   1:  PR[GP1:91,1] = PR[GP1:90,1] + -17.989;
   1:  PR[GP1:91,2] = PR[GP1:90,2] + 30.205;
   1:L PR[91] R[100]mm/sec CNT100;
   1:  PR[GP1:91,1] = PR[GP1:90,1] + -18.413;
   1:  PR[GP1:91,2] = PR[GP1:90,2] + 30.436;
   1:L PR[91] R[100]mm/sec CNT100;
   1:  PR[GP1:91,1] = PR[GP1:90,1] + -21.527;
   1:  PR[GP1:91,2] = PR[GP1:90,2] + 31.534;
   1:L PR[91] R[100]mm/sec CNT100;
   1:  PR[GP1:91,1] = PR[GP1:90,1] + -27.972;
   1:  PR[GP1:91,2] = PR[GP1:90,2] + 33.984;
   1:L PR[91] R[100]mm/sec CNT100;
   1:  PR[GP1:91,1] = PR[GP1:90,1] + -29.804;
   1:  PR[GP1:91,2] = PR[GP1:90,2] + 34.252;
   1:L PR[91] R[100]mm/sec CNT100;
   1:  PR[GP1:91,1] = PR[GP1:90,1] + -38.220;
   1:  PR[GP1:91,2] = PR[GP1:90,2] + 34.851;
   1:L PR[91] R[100]mm/sec CNT100;
   1:  PR[GP1:91,1] = PR[GP1:90,1] + -42.725;
   1:  PR[GP1:91,2] = PR[GP1:90,2] + 34.125;
   1:L PR[91] R[100]mm/sec CNT100;
   1:  PR[GP1:91,1] = PR[GP1:90,1] + -48.549;
   1:  PR[GP1:91,2] = PR[GP1:90,2] + 32.821;
   1:L PR[91] R[100]mm/sec CNT100;
   1:  PR[GP1:91,1] = PR[GP1:90,1] + -54.597;
   1:  PR[GP1:91,2] = PR[GP1:90,2] + 29.779;
   1:L PR[91] R[100]mm/sec CNT100;
   1:  PR[GP1:91,1] = PR[GP1:90,1] + -58.020;
   1:  PR[GP1:91,2] = PR[GP1:90,2] + 27.850;
   1:L PR[91] R[100]mm/sec CNT100;
   1:  PR[GP1:91,1] = PR[GP1:90,1] + -63.964;
   1:  PR[GP1:91,2] = PR[GP1:90,2] + 22.018;
   1:L PR[91] R[100]mm/sec CNT100;
   1:  PR[GP1:91,1] = PR[GP1:90,1] + -65.659;
   1:  PR[GP1:91,2] = PR[GP1:90,2] + 20.232;
   1:L PR[91] R[100]mm/sec CNT100;
   1:  PR[GP1:91,1] = PR[GP1:90,1] + -69.924;
   1:  PR[GP1:91,2] = PR[GP1:90,2] + 12.041;
   1:L PR[91] R[100]mm/sec CNT100;
   1:  PR[GP1:91,1] = PR[GP1:90,1] + -70.625;
   1:  PR[GP1:91,2] = PR[GP1:90,2] + 10.622;
   1:L PR[91] R[100]mm/sec CNT100;
   1:  PR[GP1:91,1] = PR[GP1:90,1] + -72.166;
   1:  PR[GP1:91,2] = PR[GP1:90,2] + 1.121;
   1:L PR[91] R[100]mm/sec CNT100;
   1:  PR[GP1:91,1] = PR[GP1:90,1] + -72.349;
   1:  PR[GP1:91,2] = PR[GP1:90,2] + 0.185;
   1:L PR[91] R[100]mm/sec CNT100;
   1:  PR[GP1:91,1] = PR[GP1:90,1] + -72.388;
   1:  PR[GP1:91,2] = PR[GP1:90,2] + -0.068;
   1:L PR[91] R[100]mm/sec CNT100;
   1:  PR[GP1:91,1] = PR[GP1:90,1] + -70.833;
   1:  PR[GP1:91,2] = PR[GP1:90,2] + -9.400;
   1:L PR[91] R[100]mm/sec CNT100;
   1:  PR[GP1:91,1] = PR[GP1:90,1] + -70.624;
   1:  PR[GP1:91,2] = PR[GP1:90,2] + -10.769;
   1:L PR[91] R[100]mm/sec CNT100;
   1:  PR[GP1:91,1] = PR[GP1:90,1] + -69.924;
   1:  PR[GP1:91,2] = PR[GP1:90,2] + -12.185;
   1:L PR[91] R[100]mm/sec CNT100;
   1:  PR[GP1:91,1] = PR[GP1:90,1] + -65.659;
   1:  PR[GP1:91,2] = PR[GP1:90,2] + -20.376;
   1:L PR[91] R[100]mm/sec CNT100;
   1:  PR[GP1:91,1] = PR[GP1:90,1] + -63.964;
   1:  PR[GP1:91,2] = PR[GP1:90,2] + -22.162;
   1:L PR[91] R[100]mm/sec CNT100;
   1:  PR[GP1:91,1] = PR[GP1:90,1] + -58.020;
   1:  PR[GP1:91,2] = PR[GP1:90,2] + -27.994;
   1:L PR[91] R[100]mm/sec CNT100;
   1:  PR[GP1:91,1] = PR[GP1:90,1] + -54.598;
   1:  PR[GP1:91,2] = PR[GP1:90,2] + -29.923;
   1:L PR[91] R[100]mm/sec CNT100;
   1:  PR[GP1:91,1] = PR[GP1:90,1] + -48.549;
   1:  PR[GP1:91,2] = PR[GP1:90,2] + -32.965;
   1:L PR[91] R[100]mm/sec CNT100;
   1:  PR[GP1:91,1] = PR[GP1:90,1] + -42.725;
   1:  PR[GP1:91,2] = PR[GP1:90,2] + -34.269;
   1:L PR[91] R[100]mm/sec CNT100;
   1:  PR[GP1:91,1] = PR[GP1:90,1] + -38.220;
   1:  PR[GP1:91,2] = PR[GP1:90,2] + -34.995;
   1:L PR[91] R[100]mm/sec CNT100;
   1:  PR[GP1:91,1] = PR[GP1:90,1] + -29.804;
   1:  PR[GP1:91,2] = PR[GP1:90,2] + -34.396;
   1:L PR[91] R[100]mm/sec CNT100;
   1:  PR[GP1:91,1] = PR[GP1:90,1] + -27.972;
   1:  PR[GP1:91,2] = PR[GP1:90,2] + -34.128;
   1:L PR[91] R[100]mm/sec CNT100;
   1:  PR[GP1:91,1] = PR[GP1:90,1] + -21.528;
   1:  PR[GP1:91,2] = PR[GP1:90,2] + -31.678;
   1:L PR[91] R[100]mm/sec CNT100;
   1:  PR[GP1:91,1] = PR[GP1:90,1] + -18.740;
   1:  PR[GP1:91,2] = PR[GP1:90,2] + -30.681;
   1:L PR[91] R[100]mm/sec CNT100;
   1:  PR[GP1:91,1] = PR[GP1:90,1] + -18.404;
   1:  PR[GP1:91,2] = PR[GP1:90,2] + -30.575;
   1:L PR[91] R[100]mm/sec CNT100;
   1:  PR[GP1:91,1] = PR[GP1:90,1] + -17.980;
   1:  PR[GP1:91,2] = PR[GP1:90,2] + -30.344;
   1:L PR[91] R[100]mm/sec CNT100;
   1:  PR[GP1:91,1] = PR[GP1:90,1] + -10.995;
   1:  PR[GP1:91,2] = PR[GP1:90,2] + -25.228;
   1:L PR[91] R[100]mm/sec CNT100;
   1:  PR[GP1:91,1] = PR[GP1:90,1] + -9.661;
   1:  PR[GP1:91,2] = PR[GP1:90,2] + -24.165;
   1:L PR[91] R[100]mm/sec CNT100;
   1:  PR[GP1:91,1] = PR[GP1:90,1] + -8.131;
   1:  PR[GP1:91,2] = PR[GP1:90,2] + -22.375;
   1:L PR[91] R[100]mm/sec CNT100;
   1:  PR[GP1:91,1] = PR[GP1:90,1] + -4.379;
   1:  PR[GP1:91,2] = PR[GP1:90,2] + -17.244;
   1:L PR[91] R[100]mm/sec CNT100;
   1:  PR[GP1:91,1] = PR[GP1:90,1] + -3.270;
   1:  PR[GP1:91,2] = PR[GP1:90,2] + -16.000;
   1:L PR[91] R[100]mm/sec CNT100;
   1:  PR[GP1:91,1] = PR[GP1:90,1] + -0.890;
   1:  PR[GP1:91,2] = PR[GP1:90,2] + -14.608;
   1:L PR[91] R[100]mm/sec CNT100;
   1:  PR[GP1:91,1] = PR[GP1:90,1] + 1.188;
   1:  PR[GP1:91,2] = PR[GP1:90,2] + -14.588;
   1:L PR[91] R[100]mm/sec CNT100;
   1:  PR[GP1:91,1] = PR[GP1:90,1] + 2.244;
   1:  PR[GP1:91,2] = PR[GP1:90,2] + -15.853;
   1:L PR[91] R[100]mm/sec CNT100;
   1:  PR[GP1:91,1] = PR[GP1:90,1] + 2.804;
   1:  PR[GP1:91,2] = PR[GP1:90,2] + -16.205;
   1:L PR[91] R[100]mm/sec CNT100;
   1:  PR[GP1:91,1] = PR[GP1:90,1] + 4.535;
   1:  PR[GP1:91,2] = PR[GP1:90,2] + -17.154;
   1:L PR[91] R[100]mm/sec CNT100;
   1:  PR[GP1:91,1] = PR[GP1:90,1] + 8.351;
   1:  PR[GP1:91,2] = PR[GP1:90,2] + -22.374;
   1:L PR[91] R[100]mm/sec CNT100;
   1:  PR[GP1:91,1] = PR[GP1:90,1] + 9.884;
   1:  PR[GP1:91,2] = PR[GP1:90,2] + -24.170;
   1:L PR[91] R[100]mm/sec CNT100;
   1:  PR[GP1:91,1] = PR[GP1:90,1] + 17.583;
   1:  PR[GP1:91,2] = PR[GP1:90,2] + -29.869;
   1:L PR[91] R[100]mm/sec CNT100;
   1:  PR[GP1:91,1] = PR[GP1:90,1] + 18.204;
   1:  PR[GP1:91,2] = PR[GP1:90,2] + -30.354;
   1:L PR[91] R[100]mm/sec CNT100;
   1:  PR[GP1:91,1] = PR[GP1:90,1] + 18.624;
   1:  PR[GP1:91,2] = PR[GP1:90,2] + -30.582;
   1:L PR[91] R[100]mm/sec CNT100;
   1:  PR[GP1:91,1] = PR[GP1:90,1] + 21.740;
   1:  PR[GP1:91,2] = PR[GP1:90,2] + -31.680;
   1:L PR[91] R[100]mm/sec CNT100;
   1:  PR[GP1:91,1] = PR[GP1:90,1] + 28.183;
   1:  PR[GP1:91,2] = PR[GP1:90,2] + -34.126;
   1:L PR[91] R[100]mm/sec CNT100;
   1:  PR[GP1:91,1] = PR[GP1:90,1] + 30.015;
   1:  PR[GP1:91,2] = PR[GP1:90,2] + -34.395;
   1:L PR[91] R[100]mm/sec CNT100;
   1:  PR[GP1:91,1] = PR[GP1:90,1] + 38.429;
   1:  PR[GP1:91,2] = PR[GP1:90,2] + -34.995;
   1:L PR[91] R[100]mm/sec CNT100;
   1:  PR[GP1:91,1] = PR[GP1:90,1] + 42.934;
   1:  PR[GP1:91,2] = PR[GP1:90,2] + -34.270;
   1:L PR[91] R[100]mm/sec CNT100;
   1:  PR[GP1:91,1] = PR[GP1:90,1] + 48.758;
   1:  PR[GP1:91,2] = PR[GP1:90,2] + -32.964;
   1:L PR[91] R[100]mm/sec CNT100;
   1:  PR[GP1:91,1] = PR[GP1:90,1] + 54.807;
   1:  PR[GP1:91,2] = PR[GP1:90,2] + -29.927;
   1:L PR[91] R[100]mm/sec CNT100;
   1:  PR[GP1:91,1] = PR[GP1:90,1] + 58.229;
   1:  PR[GP1:91,2] = PR[GP1:90,2] + -28.001;
   1:L PR[91] R[100]mm/sec CNT100;
   1:  PR[GP1:91,1] = PR[GP1:90,1] + 64.175;
   1:  PR[GP1:91,2] = PR[GP1:90,2] + -22.159;
   1:L PR[91] R[100]mm/sec CNT100;
   1:  PR[GP1:91,1] = PR[GP1:90,1] + 65.870;
   1:  PR[GP1:91,2] = PR[GP1:90,2] + -20.368;
   1:L PR[91] R[100]mm/sec CNT100;
   1:  PR[GP1:91,1] = PR[GP1:90,1] + 70.137;
   1:  PR[GP1:91,2] = PR[GP1:90,2] + -12.197;
   1:L PR[91] R[100]mm/sec CNT100;
   1:  PR[GP1:91,1] = PR[GP1:90,1] + 70.838;
   1:  PR[GP1:91,2] = PR[GP1:90,2] + -10.785;
   1:L PR[91] R[100]mm/sec CNT100;
   1:  PR[GP1:91,1] = PR[GP1:90,1] + 72.380;
   1:  PR[GP1:91,2] = PR[GP1:90,2] + -1.269;
   1:L PR[91] R[100]mm/sec CNT100;
   1:  PR[GP1:91,1] = PR[GP1:90,1] + 72.563;
   1:  PR[GP1:91,2] = PR[GP1:90,2] + -0.331;
   1:L PR[91] R[100]mm/sec CNT100;
   1:  PR[GP1:91,1] = PR[GP1:90,1] + 72.601;
   1:  PR[GP1:91,2] = PR[GP1:90,2] + -0.076;
   1:L PR[91] R[100]mm/sec CNT100;
   1:  PR[GP1:91,1] = PR[GP1:90,1] + 71.045;
   1:  PR[GP1:91,2] = PR[GP1:90,2] + 9.272;
   1:L PR[91] R[100]mm/sec CNT100;
   1:  PR[GP1:91,1] = PR[GP1:90,1] + 70.837;
   1:  PR[GP1:91,2] = PR[GP1:90,2] + 10.644;
   1:L PR[91] R[100]mm/sec CNT100;
   1:  PR[GP1:91,1] = PR[GP1:90,1] + 70.137;
   1:  PR[GP1:91,2] = PR[GP1:90,2] + 12.053;
   1:L PR[91] R[100]mm/sec CNT100;
   1:  PR[GP1:91,1] = PR[GP1:90,1] + 65.870;
   1:  PR[GP1:91,2] = PR[GP1:90,2] + 20.224;
   1:L PR[91] R[100]mm/sec CNT100;
   1:  PR[GP1:91,1] = PR[GP1:90,1] + 64.175;
   1:  PR[GP1:91,2] = PR[GP1:90,2] + 22.015;
   1:L PR[91] R[100]mm/sec CNT100;
   1:  PR[GP1:91,1] = PR[GP1:90,1] + 58.229;
   1:  PR[GP1:91,2] = PR[GP1:90,2] + 27.857;
   1:L PR[91] R[100]mm/sec CNT100;
   1:  PR[GP1:91,1] = PR[GP1:90,1] + 54.807;
   1:  PR[GP1:91,2] = PR[GP1:90,2] + 29.783;
   1:L PR[91] R[100]mm/sec CNT100;
   1:  PR[GP1:91,1] = PR[GP1:90,1] + 48.758;
   1:  PR[GP1:91,2] = PR[GP1:90,2] + 32.820;
   1:L PR[91] R[100]mm/sec CNT100;
   1:  PR[GP1:91,1] = PR[GP1:90,1] + 42.934;
   1:  PR[GP1:91,2] = PR[GP1:90,2] + 34.126;
   1:L PR[91] R[100]mm/sec CNT100;
   1:  PR[GP1:91,1] = PR[GP1:90,1] + 38.429;
   1:  PR[GP1:91,2] = PR[GP1:90,2] + 34.851;
   1:L PR[91] R[100]mm/sec CNT100;
   1:  PR[GP1:91,1] = PR[GP1:90,1] + 30.015;
   1:  PR[GP1:91,2] = PR[GP1:90,2] + 34.251;
   1:L PR[91] R[100]mm/sec CNT100;
   1:  PR[GP1:91,1] = PR[GP1:90,1] + 28.183;
   1:  PR[GP1:91,2] = PR[GP1:90,2] + 33.982;
   1:L PR[91] R[100]mm/sec CNT100;
   1:  PR[GP1:91,1] = PR[GP1:90,1] + 21.741;
   1:  PR[GP1:91,2] = PR[GP1:90,2] + 31.536;
   1:L PR[91] R[100]mm/sec CNT100;
   1:  PR[GP1:91,1] = PR[GP1:90,1] + 18.953;
   1:  PR[GP1:91,2] = PR[GP1:90,2] + 30.540;
   1:L PR[91] R[100]mm/sec CNT100;
   1:  PR[GP1:91,1] = PR[GP1:90,1] + 18.616;
   1:  PR[GP1:91,2] = PR[GP1:90,2] + 30.434;
   1:L PR[91] R[100]mm/sec CNT100;
   1:  PR[GP1:91,1] = PR[GP1:90,1] + 18.196;
   1:  PR[GP1:91,2] = PR[GP1:90,2] + 30.205;
   1:L PR[91] R[100]mm/sec CNT100;
   1:  PR[GP1:91,1] = PR[GP1:90,1] + 11.213;
   1:  PR[GP1:91,2] = PR[GP1:90,2] + 25.087;
   1:L PR[91] R[100]mm/sec CNT100;
   1:  PR[GP1:91,1] = PR[GP1:90,1] + 9.890;
   1:  PR[GP1:91,2] = PR[GP1:90,2] + 24.034;
   1:L PR[91] R[100]mm/sec CNT100;
   1:  PR[GP1:91,1] = PR[GP1:90,1] + 8.351;
   1:  PR[GP1:91,2] = PR[GP1:90,2] + 22.230;
   1:L PR[91] R[100]mm/sec CNT100;
   1:  PR[GP1:91,1] = PR[GP1:90,1] + 4.595;
   1:  PR[GP1:91,2] = PR[GP1:90,2] + 17.092;
   1:L PR[91] R[100]mm/sec CNT100;
   1:  PR[GP1:91,1] = PR[GP1:90,1] + 3.455;
   1:  PR[GP1:91,2] = PR[GP1:90,2] + 15.837;
   1:L PR[91] R[100]mm/sec CNT100;
   1:  PR[GP1:91,1] = PR[GP1:90,1] + 1.069;
   1:  PR[GP1:91,2] = PR[GP1:90,2] + 14.445;
   1:L PR[91] R[100]mm/sec CNT100;
   1:  PR[GP1:91,1] = PR[GP1:90,1] + -0.890;
   1:  PR[GP1:91,2] = PR[GP1:90,2] + 14.464;
   1:L PR[91] R[100]mm/sec CNT100;
   1:  ! -- Layer/Ebene 55 -- !;
   1:  PR[91] = PR[90];
   1:  PR[GP1:91,1] = PR[GP1:90,1] + -3.388;
   1:  PR[GP1:91,2] = PR[GP1:90,2] + 16.407;
   1:  PR[GP1:91,3] = PR[GP1:90,3] + 33.855;
   1:L PR[91] R[100]mm/sec CNT100;
   1:  PR[GP1:91,1] = PR[GP1:90,1] + -4.446;
   1:  PR[GP1:91,2] = PR[GP1:90,2] + 17.549;
   1:L PR[91] R[100]mm/sec CNT100;
   1:  PR[GP1:91,1] = PR[GP1:90,1] + -4.455;
   1:  PR[GP1:91,2] = PR[GP1:90,2] + 17.629;
   1:L PR[91] R[100]mm/sec CNT100;
   1:  PR[GP1:91,1] = PR[GP1:90,1] + -7.518;
   1:  PR[GP1:91,2] = PR[GP1:90,2] + 21.818;
   1:L PR[91] R[100]mm/sec CNT100;
   1:  PR[GP1:91,1] = PR[GP1:90,1] + -9.459;
   1:  PR[GP1:91,2] = PR[GP1:90,2] + 24.089;
   1:L PR[91] R[100]mm/sec CNT100;
   1:  PR[GP1:91,1] = PR[GP1:90,1] + -16.227;
   1:  PR[GP1:91,2] = PR[GP1:90,2] + 29.096;
   1:L PR[91] R[100]mm/sec CNT100;
   1:  PR[GP1:91,1] = PR[GP1:90,1] + -17.485;
   1:  PR[GP1:91,2] = PR[GP1:90,2] + 30.078;
   1:L PR[91] R[100]mm/sec CNT100;
   1:  PR[GP1:91,1] = PR[GP1:90,1] + -18.396;
   1:  PR[GP1:91,2] = PR[GP1:90,2] + 30.575;
   1:L PR[91] R[100]mm/sec CNT100;
   1:  PR[GP1:91,1] = PR[GP1:90,1] + -24.522;
   1:  PR[GP1:91,2] = PR[GP1:90,2] + 32.735;
   1:L PR[91] R[100]mm/sec CNT100;
   1:  PR[GP1:91,1] = PR[GP1:90,1] + -28.037;
   1:  PR[GP1:91,2] = PR[GP1:90,2] + 34.071;
   1:L PR[91] R[100]mm/sec CNT100;
   1:  PR[GP1:91,1] = PR[GP1:90,1] + -29.004;
   1:  PR[GP1:91,2] = PR[GP1:90,2] + 34.213;
   1:L PR[91] R[100]mm/sec CNT100;
   1:  PR[GP1:91,1] = PR[GP1:90,1] + -38.254;
   1:  PR[GP1:91,2] = PR[GP1:90,2] + 34.871;
   1:L PR[91] R[100]mm/sec CNT100;
   1:  PR[GP1:91,1] = PR[GP1:90,1] + -41.956;
   1:  PR[GP1:91,2] = PR[GP1:90,2] + 34.274;
   1:L PR[91] R[100]mm/sec CNT100;
   1:  PR[GP1:91,1] = PR[GP1:90,1] + -48.542;
   1:  PR[GP1:91,2] = PR[GP1:90,2] + 32.799;
   1:L PR[91] R[100]mm/sec CNT100;
   1:  PR[GP1:91,1] = PR[GP1:90,1] + -53.920;
   1:  PR[GP1:91,2] = PR[GP1:90,2] + 30.095;
   1:L PR[91] R[100]mm/sec CNT100;
   1:  PR[GP1:91,1] = PR[GP1:90,1] + -57.970;
   1:  PR[GP1:91,2] = PR[GP1:90,2] + 27.812;
   1:L PR[91] R[100]mm/sec CNT100;
   1:  PR[GP1:91,1] = PR[GP1:90,1] + -63.421;
   1:  PR[GP1:91,2] = PR[GP1:90,2] + 22.463;
   1:L PR[91] R[100]mm/sec CNT100;
   1:  PR[GP1:91,1] = PR[GP1:90,1] + -65.574;
   1:  PR[GP1:91,2] = PR[GP1:90,2] + 20.196;
   1:L PR[91] R[100]mm/sec CNT100;
   1:  PR[GP1:91,1] = PR[GP1:90,1] + -69.543;
   1:  PR[GP1:91,2] = PR[GP1:90,2] + 12.572;
   1:L PR[91] R[100]mm/sec CNT100;
   1:  PR[GP1:91,1] = PR[GP1:90,1] + -70.517;
   1:  PR[GP1:91,2] = PR[GP1:90,2] + 10.601;
   1:L PR[91] R[100]mm/sec CNT100;
   1:  PR[GP1:91,1] = PR[GP1:90,1] + -71.962;
   1:  PR[GP1:91,2] = PR[GP1:90,2] + 1.695;
   1:L PR[91] R[100]mm/sec CNT100;
   1:  PR[GP1:91,1] = PR[GP1:90,1] + -72.133;
   1:  PR[GP1:91,2] = PR[GP1:90,2] + 0.818;
   1:L PR[91] R[100]mm/sec CNT100;
   1:  PR[GP1:91,1] = PR[GP1:90,1] + -72.269;
   1:  PR[GP1:91,2] = PR[GP1:90,2] + -0.068;
   1:L PR[91] R[100]mm/sec CNT100;
   1:  PR[GP1:91,1] = PR[GP1:90,1] + -70.806;
   1:  PR[GP1:91,2] = PR[GP1:90,2] + -8.846;
   1:L PR[91] R[100]mm/sec CNT100;
   1:  PR[GP1:91,1] = PR[GP1:90,1] + -70.516;
   1:  PR[GP1:91,2] = PR[GP1:90,2] + -10.748;
   1:L PR[91] R[100]mm/sec CNT100;
   1:  PR[GP1:91,1] = PR[GP1:90,1] + -69.543;
   1:  PR[GP1:91,2] = PR[GP1:90,2] + -12.716;
   1:L PR[91] R[100]mm/sec CNT100;
   1:  PR[GP1:91,1] = PR[GP1:90,1] + -65.574;
   1:  PR[GP1:91,2] = PR[GP1:90,2] + -20.340;
   1:L PR[91] R[100]mm/sec CNT100;
   1:  PR[GP1:91,1] = PR[GP1:90,1] + -63.421;
   1:  PR[GP1:91,2] = PR[GP1:90,2] + -22.607;
   1:L PR[91] R[100]mm/sec CNT100;
   1:  PR[GP1:91,1] = PR[GP1:90,1] + -57.970;
   1:  PR[GP1:91,2] = PR[GP1:90,2] + -27.956;
   1:L PR[91] R[100]mm/sec CNT100;
   1:  PR[GP1:91,1] = PR[GP1:90,1] + -53.920;
   1:  PR[GP1:91,2] = PR[GP1:90,2] + -30.239;
   1:L PR[91] R[100]mm/sec CNT100;
   1:  PR[GP1:91,1] = PR[GP1:90,1] + -48.542;
   1:  PR[GP1:91,2] = PR[GP1:90,2] + -32.943;
   1:L PR[91] R[100]mm/sec CNT100;
   1:  PR[GP1:91,1] = PR[GP1:90,1] + -41.956;
   1:  PR[GP1:91,2] = PR[GP1:90,2] + -34.418;
   1:L PR[91] R[100]mm/sec CNT100;
   1:  PR[GP1:91,1] = PR[GP1:90,1] + -38.254;
   1:  PR[GP1:91,2] = PR[GP1:90,2] + -35.015;
   1:L PR[91] R[100]mm/sec CNT100;
   1:  PR[GP1:91,1] = PR[GP1:90,1] + -29.004;
   1:  PR[GP1:91,2] = PR[GP1:90,2] + -34.357;
   1:L PR[91] R[100]mm/sec CNT100;
   1:  PR[GP1:91,1] = PR[GP1:90,1] + -28.037;
   1:  PR[GP1:91,2] = PR[GP1:90,2] + -34.215;
   1:L PR[91] R[100]mm/sec CNT100;
   1:  PR[GP1:91,1] = PR[GP1:90,1] + -24.523;
   1:  PR[GP1:91,2] = PR[GP1:90,2] + -32.879;
   1:L PR[91] R[100]mm/sec CNT100;
   1:  PR[GP1:91,1] = PR[GP1:90,1] + -19.087;
   1:  PR[GP1:91,2] = PR[GP1:90,2] + -30.934;
   1:L PR[91] R[100]mm/sec CNT100;
   1:  PR[GP1:91,1] = PR[GP1:90,1] + -18.387;
   1:  PR[GP1:91,2] = PR[GP1:90,2] + -30.714;
   1:L PR[91] R[100]mm/sec CNT100;
   1:  PR[GP1:91,1] = PR[GP1:90,1] + -17.476;
   1:  PR[GP1:91,2] = PR[GP1:90,2] + -30.217;
   1:L PR[91] R[100]mm/sec CNT100;
   1:  PR[GP1:91,1] = PR[GP1:90,1] + -11.167;
   1:  PR[GP1:91,2] = PR[GP1:90,2] + -25.597;
   1:L PR[91] R[100]mm/sec CNT100;
   1:  PR[GP1:91,1] = PR[GP1:90,1] + -9.466;
   1:  PR[GP1:91,2] = PR[GP1:90,2] + -24.241;
   1:L PR[91] R[100]mm/sec CNT100;
   1:  PR[GP1:91,1] = PR[GP1:90,1] + -7.518;
   1:  PR[GP1:91,2] = PR[GP1:90,2] + -21.962;
   1:L PR[91] R[100]mm/sec CNT100;
   1:  PR[GP1:91,1] = PR[GP1:90,1] + -4.344;
   1:  PR[GP1:91,2] = PR[GP1:90,2] + -17.621;
   1:L PR[91] R[100]mm/sec CNT100;
   1:  PR[GP1:91,1] = PR[GP1:90,1] + -3.393;
   1:  PR[GP1:91,2] = PR[GP1:90,2] + -16.554;
   1:L PR[91] R[100]mm/sec CNT100;
   1:  PR[GP1:91,1] = PR[GP1:90,1] + -0.787;
   1:  PR[GP1:91,2] = PR[GP1:90,2] + -15.030;
   1:L PR[91] R[100]mm/sec CNT100;
   1:  PR[GP1:91,1] = PR[GP1:90,1] + 1.090;
   1:  PR[GP1:91,2] = PR[GP1:90,2] + -15.011;
   1:L PR[91] R[100]mm/sec CNT100;
   1:  PR[GP1:91,1] = PR[GP1:90,1] + 2.030;
   1:  PR[GP1:91,2] = PR[GP1:90,2] + -16.138;
   1:L PR[91] R[100]mm/sec CNT100;
   1:  PR[GP1:91,1] = PR[GP1:90,1] + 2.509;
   1:  PR[GP1:91,2] = PR[GP1:90,2] + -16.440;
   1:L PR[91] R[100]mm/sec CNT100;
   1:  PR[GP1:91,1] = PR[GP1:90,1] + 4.501;
   1:  PR[GP1:91,2] = PR[GP1:90,2] + -17.531;
   1:L PR[91] R[100]mm/sec CNT100;
   1:  PR[GP1:91,1] = PR[GP1:90,1] + 7.740;
   1:  PR[GP1:91,2] = PR[GP1:90,2] + -21.961;
   1:L PR[91] R[100]mm/sec CNT100;
   1:  PR[GP1:91,1] = PR[GP1:90,1] + 9.693;
   1:  PR[GP1:91,2] = PR[GP1:90,2] + -24.250;
   1:L PR[91] R[100]mm/sec CNT100;
   1:  PR[GP1:91,1] = PR[GP1:90,1] + 16.456;
   1:  PR[GP1:91,2] = PR[GP1:90,2] + -29.256;
   1:L PR[91] R[100]mm/sec CNT100;
   1:  PR[GP1:91,1] = PR[GP1:90,1] + 17.702;
   1:  PR[GP1:91,2] = PR[GP1:90,2] + -30.229;
   1:L PR[91] R[100]mm/sec CNT100;
   1:  PR[GP1:91,1] = PR[GP1:90,1] + 18.606;
   1:  PR[GP1:91,2] = PR[GP1:90,2] + -30.721;
   1:L PR[91] R[100]mm/sec CNT100;
   1:  PR[GP1:91,1] = PR[GP1:90,1] + 24.735;
   1:  PR[GP1:91,2] = PR[GP1:90,2] + -32.879;
   1:L PR[91] R[100]mm/sec CNT100;
   1:  PR[GP1:91,1] = PR[GP1:90,1] + 28.250;
   1:  PR[GP1:91,2] = PR[GP1:90,2] + -34.213;
   1:L PR[91] R[100]mm/sec CNT100;
   1:  PR[GP1:91,1] = PR[GP1:90,1] + 29.217;
   1:  PR[GP1:91,2] = PR[GP1:90,2] + -34.355;
   1:L PR[91] R[100]mm/sec CNT100;
   1:  PR[GP1:91,1] = PR[GP1:90,1] + 38.464;
   1:  PR[GP1:91,2] = PR[GP1:90,2] + -35.015;
   1:L PR[91] R[100]mm/sec CNT100;
   1:  PR[GP1:91,1] = PR[GP1:90,1] + 42.166;
   1:  PR[GP1:91,2] = PR[GP1:90,2] + -34.419;
   1:L PR[91] R[100]mm/sec CNT100;
   1:  PR[GP1:91,1] = PR[GP1:90,1] + 48.751;
   1:  PR[GP1:91,2] = PR[GP1:90,2] + -32.942;
   1:L PR[91] R[100]mm/sec CNT100;
   1:  PR[GP1:91,1] = PR[GP1:90,1] + 54.129;
   1:  PR[GP1:91,2] = PR[GP1:90,2] + -30.242;
   1:L PR[91] R[100]mm/sec CNT100;
   1:  PR[GP1:91,1] = PR[GP1:90,1] + 58.179;
   1:  PR[GP1:91,2] = PR[GP1:90,2] + -27.963;
   1:L PR[91] R[100]mm/sec CNT100;
   1:  PR[GP1:91,1] = PR[GP1:90,1] + 63.632;
   1:  PR[GP1:91,2] = PR[GP1:90,2] + -22.606;
   1:L PR[91] R[100]mm/sec CNT100;
   1:  PR[GP1:91,1] = PR[GP1:90,1] + 65.785;
   1:  PR[GP1:91,2] = PR[GP1:90,2] + -20.331;
   1:L PR[91] R[100]mm/sec CNT100;
   1:  PR[GP1:91,1] = PR[GP1:90,1] + 69.756;
   1:  PR[GP1:91,2] = PR[GP1:90,2] + -12.726;
   1:L PR[91] R[100]mm/sec CNT100;
   1:  PR[GP1:91,1] = PR[GP1:90,1] + 70.730;
   1:  PR[GP1:91,2] = PR[GP1:90,2] + -10.765;
   1:L PR[91] R[100]mm/sec CNT100;
   1:  PR[GP1:91,1] = PR[GP1:90,1] + 72.175;
   1:  PR[GP1:91,2] = PR[GP1:90,2] + -1.845;
   1:L PR[91] R[100]mm/sec CNT100;
   1:  PR[GP1:91,1] = PR[GP1:90,1] + 72.346;
   1:  PR[GP1:91,2] = PR[GP1:90,2] + -0.965;
   1:L PR[91] R[100]mm/sec CNT100;
   1:  PR[GP1:91,1] = PR[GP1:90,1] + 72.482;
   1:  PR[GP1:91,2] = PR[GP1:90,2] + -0.076;
   1:L PR[91] R[100]mm/sec CNT100;
   1:  PR[GP1:91,1] = PR[GP1:90,1] + 71.019;
   1:  PR[GP1:91,2] = PR[GP1:90,2] + 8.717;
   1:L PR[91] R[100]mm/sec CNT100;
   1:  PR[GP1:91,1] = PR[GP1:90,1] + 70.728;
   1:  PR[GP1:91,2] = PR[GP1:90,2] + 10.624;
   1:L PR[91] R[100]mm/sec CNT100;
   1:  PR[GP1:91,1] = PR[GP1:90,1] + 69.756;
   1:  PR[GP1:91,2] = PR[GP1:90,2] + 12.582;
   1:L PR[91] R[100]mm/sec CNT100;
   1:  PR[GP1:91,1] = PR[GP1:90,1] + 65.785;
   1:  PR[GP1:91,2] = PR[GP1:90,2] + 20.187;
   1:L PR[91] R[100]mm/sec CNT100;
   1:  PR[GP1:91,1] = PR[GP1:90,1] + 63.632;
   1:  PR[GP1:91,2] = PR[GP1:90,2] + 22.462;
   1:L PR[91] R[100]mm/sec CNT100;
   1:  PR[GP1:91,1] = PR[GP1:90,1] + 58.179;
   1:  PR[GP1:91,2] = PR[GP1:90,2] + 27.819;
   1:L PR[91] R[100]mm/sec CNT100;
   1:  PR[GP1:91,1] = PR[GP1:90,1] + 54.129;
   1:  PR[GP1:91,2] = PR[GP1:90,2] + 30.098;
   1:L PR[91] R[100]mm/sec CNT100;
   1:  PR[GP1:91,1] = PR[GP1:90,1] + 48.751;
   1:  PR[GP1:91,2] = PR[GP1:90,2] + 32.798;
   1:L PR[91] R[100]mm/sec CNT100;
   1:  PR[GP1:91,1] = PR[GP1:90,1] + 42.166;
   1:  PR[GP1:91,2] = PR[GP1:90,2] + 34.275;
   1:L PR[91] R[100]mm/sec CNT100;
   1:  PR[GP1:91,1] = PR[GP1:90,1] + 38.464;
   1:  PR[GP1:91,2] = PR[GP1:90,2] + 34.871;
   1:L PR[91] R[100]mm/sec CNT100;
   1:  PR[GP1:91,1] = PR[GP1:90,1] + 29.217;
   1:  PR[GP1:91,2] = PR[GP1:90,2] + 34.211;
   1:L PR[91] R[100]mm/sec CNT100;
   1:  PR[GP1:91,1] = PR[GP1:90,1] + 28.250;
   1:  PR[GP1:91,2] = PR[GP1:90,2] + 34.069;
   1:L PR[91] R[100]mm/sec CNT100;
   1:  PR[GP1:91,1] = PR[GP1:90,1] + 24.736;
   1:  PR[GP1:91,2] = PR[GP1:90,2] + 32.735;
   1:L PR[91] R[100]mm/sec CNT100;
   1:  PR[GP1:91,1] = PR[GP1:90,1] + 19.300;
   1:  PR[GP1:91,2] = PR[GP1:90,2] + 30.793;
   1:L PR[91] R[100]mm/sec CNT100;
   1:  PR[GP1:91,1] = PR[GP1:90,1] + 18.598;
   1:  PR[GP1:91,2] = PR[GP1:90,2] + 30.572;
   1:L PR[91] R[100]mm/sec CNT100;
   1:  PR[GP1:91,1] = PR[GP1:90,1] + 17.694;
   1:  PR[GP1:91,2] = PR[GP1:90,2] + 30.080;
   1:L PR[91] R[100]mm/sec CNT100;
   1:  PR[GP1:91,1] = PR[GP1:90,1] + 11.387;
   1:  PR[GP1:91,2] = PR[GP1:90,2] + 25.457;
   1:L PR[91] R[100]mm/sec CNT100;
   1:  PR[GP1:91,1] = PR[GP1:90,1] + 9.700;
   1:  PR[GP1:91,2] = PR[GP1:90,2] + 24.114;
   1:L PR[91] R[100]mm/sec CNT100;
   1:  PR[GP1:91,1] = PR[GP1:90,1] + 7.740;
   1:  PR[GP1:91,2] = PR[GP1:90,2] + 21.817;
   1:L PR[91] R[100]mm/sec CNT100;
   1:  PR[GP1:91,1] = PR[GP1:90,1] + 4.561;
   1:  PR[GP1:91,2] = PR[GP1:90,2] + 17.469;
   1:L PR[91] R[100]mm/sec CNT100;
   1:  PR[GP1:91,1] = PR[GP1:90,1] + 3.583;
   1:  PR[GP1:91,2] = PR[GP1:90,2] + 16.393;
   1:L PR[91] R[100]mm/sec CNT100;
   1:  PR[GP1:91,1] = PR[GP1:90,1] + 0.971;
   1:  PR[GP1:91,2] = PR[GP1:90,2] + 14.869;
   1:L PR[91] R[100]mm/sec CNT100;
   1:  PR[GP1:91,1] = PR[GP1:90,1] + -0.787;
   1:  PR[GP1:91,2] = PR[GP1:90,2] + 14.886;
   1:L PR[91] R[100]mm/sec CNT100;
   1:  ! -- Layer/Ebene 56 -- !;
   1:  PR[91] = PR[90];
   1:  PR[GP1:91,1] = PR[GP1:90,1] + -3.510;
   1:  PR[GP1:91,2] = PR[GP1:90,2] + 16.961;
   1:  PR[GP1:91,3] = PR[GP1:90,3] + 34.465;
   1:L PR[91] R[100]mm/sec CNT100;
   1:  PR[GP1:91,1] = PR[GP1:90,1] + -4.411;
   1:  PR[GP1:91,2] = PR[GP1:90,2] + 17.933;
   1:L PR[91] R[100]mm/sec CNT100;
   1:  PR[GP1:91,1] = PR[GP1:90,1] + -4.420;
   1:  PR[GP1:91,2] = PR[GP1:90,2] + 18.006;
   1:L PR[91] R[100]mm/sec CNT100;
   1:  PR[GP1:91,1] = PR[GP1:90,1] + -6.905;
   1:  PR[GP1:91,2] = PR[GP1:90,2] + 21.405;
   1:L PR[91] R[100]mm/sec CNT100;
   1:  PR[GP1:91,1] = PR[GP1:90,1] + -9.264;
   1:  PR[GP1:91,2] = PR[GP1:90,2] + 24.165;
   1:L PR[91] R[100]mm/sec CNT100;
   1:  PR[GP1:91,1] = PR[GP1:90,1] + -15.093;
   1:  PR[GP1:91,2] = PR[GP1:90,2] + 28.477;
   1:L PR[91] R[100]mm/sec CNT100;
   1:  PR[GP1:91,1] = PR[GP1:90,1] + -16.981;
   1:  PR[GP1:91,2] = PR[GP1:90,2] + 29.951;
   1:L PR[91] R[100]mm/sec CNT100;
   1:  PR[GP1:91,1] = PR[GP1:90,1] + -18.379;
   1:  PR[GP1:91,2] = PR[GP1:90,2] + 30.714;
   1:L PR[91] R[100]mm/sec CNT100;
   1:  PR[GP1:91,1] = PR[GP1:90,1] + -27.518;
   1:  PR[GP1:91,2] = PR[GP1:90,2] + 33.936;
   1:L PR[91] R[100]mm/sec CNT100;
   1:  PR[GP1:91,1] = PR[GP1:90,1] + -28.103;
   1:  PR[GP1:91,2] = PR[GP1:90,2] + 34.158;
   1:L PR[91] R[100]mm/sec CNT100;
   1:  PR[GP1:91,1] = PR[GP1:90,1] + -28.204;
   1:  PR[GP1:91,2] = PR[GP1:90,2] + 34.173;
   1:L PR[91] R[100]mm/sec CNT100;
   1:  PR[GP1:91,1] = PR[GP1:90,1] + -38.288;
   1:  PR[GP1:91,2] = PR[GP1:90,2] + 34.890;
   1:L PR[91] R[100]mm/sec CNT100;
   1:  PR[GP1:91,1] = PR[GP1:90,1] + -41.188;
   1:  PR[GP1:91,2] = PR[GP1:90,2] + 34.423;
   1:L PR[91] R[100]mm/sec CNT100;
   1:  PR[GP1:91,1] = PR[GP1:90,1] + -48.534;
   1:  PR[GP1:91,2] = PR[GP1:90,2] + 32.778;
   1:L PR[91] R[100]mm/sec CNT100;
   1:  PR[GP1:91,1] = PR[GP1:90,1] + -53.242;
   1:  PR[GP1:91,2] = PR[GP1:90,2] + 30.410;
   1:L PR[91] R[100]mm/sec CNT100;
   1:  PR[GP1:91,1] = PR[GP1:90,1] + -57.919;
   1:  PR[GP1:91,2] = PR[GP1:90,2] + 27.773;
   1:L PR[91] R[100]mm/sec CNT100;
   1:  PR[GP1:91,1] = PR[GP1:90,1] + -62.878;
   1:  PR[GP1:91,2] = PR[GP1:90,2] + 22.909;
   1:L PR[91] R[100]mm/sec CNT100;
   1:  PR[GP1:91,1] = PR[GP1:90,1] + -65.489;
   1:  PR[GP1:91,2] = PR[GP1:90,2] + 20.159;
   1:L PR[91] R[100]mm/sec CNT100;
   1:  PR[GP1:91,1] = PR[GP1:90,1] + -69.163;
   1:  PR[GP1:91,2] = PR[GP1:90,2] + 13.103;
   1:L PR[91] R[100]mm/sec CNT100;
   1:  PR[GP1:91,1] = PR[GP1:90,1] + -70.409;
   1:  PR[GP1:91,2] = PR[GP1:90,2] + 10.580;
   1:L PR[91] R[100]mm/sec CNT100;
   1:  PR[GP1:91,1] = PR[GP1:90,1] + -71.757;
   1:  PR[GP1:91,2] = PR[GP1:90,2] + 2.270;
   1:L PR[91] R[100]mm/sec CNT100;
   1:  PR[GP1:91,1] = PR[GP1:90,1] + -71.917;
   1:  PR[GP1:91,2] = PR[GP1:90,2] + 1.451;
   1:L PR[91] R[100]mm/sec CNT100;
   1:  PR[GP1:91,1] = PR[GP1:90,1] + -72.150;
   1:  PR[GP1:91,2] = PR[GP1:90,2] + -0.068;
   1:L PR[91] R[100]mm/sec CNT100;
   1:  PR[GP1:91,1] = PR[GP1:90,1] + -70.779;
   1:  PR[GP1:91,2] = PR[GP1:90,2] + -8.291;
   1:L PR[91] R[100]mm/sec CNT100;
   1:  PR[GP1:91,1] = PR[GP1:90,1] + -70.407;
   1:  PR[GP1:91,2] = PR[GP1:90,2] + -10.727;
   1:L PR[91] R[100]mm/sec CNT100;
   1:  PR[GP1:91,1] = PR[GP1:90,1] + -69.163;
   1:  PR[GP1:91,2] = PR[GP1:90,2] + -13.247;
   1:L PR[91] R[100]mm/sec CNT100;
   1:  PR[GP1:91,1] = PR[GP1:90,1] + -65.489;
   1:  PR[GP1:91,2] = PR[GP1:90,2] + -20.303;
   1:L PR[91] R[100]mm/sec CNT100;
   1:  PR[GP1:91,1] = PR[GP1:90,1] + -62.878;
   1:  PR[GP1:91,2] = PR[GP1:90,2] + -23.053;
   1:L PR[91] R[100]mm/sec CNT100;
   1:  PR[GP1:91,1] = PR[GP1:90,1] + -57.919;
   1:  PR[GP1:91,2] = PR[GP1:90,2] + -27.917;
   1:L PR[91] R[100]mm/sec CNT100;
   1:  PR[GP1:91,1] = PR[GP1:90,1] + -53.242;
   1:  PR[GP1:91,2] = PR[GP1:90,2] + -30.554;
   1:L PR[91] R[100]mm/sec CNT100;
   1:  PR[GP1:91,1] = PR[GP1:90,1] + -48.534;
   1:  PR[GP1:91,2] = PR[GP1:90,2] + -32.922;
   1:L PR[91] R[100]mm/sec CNT100;
   1:  PR[GP1:91,1] = PR[GP1:90,1] + -41.188;
   1:  PR[GP1:91,2] = PR[GP1:90,2] + -34.567;
   1:L PR[91] R[100]mm/sec CNT100;
   1:  PR[GP1:91,1] = PR[GP1:90,1] + -38.288;
   1:  PR[GP1:91,2] = PR[GP1:90,2] + -35.034;
   1:L PR[91] R[100]mm/sec CNT100;
   1:  PR[GP1:91,1] = PR[GP1:90,1] + -28.204;
   1:  PR[GP1:91,2] = PR[GP1:90,2] + -34.317;
   1:L PR[91] R[100]mm/sec CNT100;
   1:  PR[GP1:91,1] = PR[GP1:90,1] + -28.103;
   1:  PR[GP1:91,2] = PR[GP1:90,2] + -34.302;
   1:L PR[91] R[100]mm/sec CNT100;
   1:  PR[GP1:91,1] = PR[GP1:90,1] + -27.519;
   1:  PR[GP1:91,2] = PR[GP1:90,2] + -34.080;
   1:L PR[91] R[100]mm/sec CNT100;
   1:  PR[GP1:91,1] = PR[GP1:90,1] + -19.434;
   1:  PR[GP1:91,2] = PR[GP1:90,2] + -31.187;
   1:L PR[91] R[100]mm/sec CNT100;
   1:  PR[GP1:91,1] = PR[GP1:90,1] + -18.370;
   1:  PR[GP1:91,2] = PR[GP1:90,2] + -30.852;
   1:L PR[91] R[100]mm/sec CNT100;
   1:  PR[GP1:91,1] = PR[GP1:90,1] + -16.973;
   1:  PR[GP1:91,2] = PR[GP1:90,2] + -30.091;
   1:L PR[91] R[100]mm/sec CNT100;
   1:  PR[GP1:91,1] = PR[GP1:90,1] + -11.340;
   1:  PR[GP1:91,2] = PR[GP1:90,2] + -25.965;
   1:L PR[91] R[100]mm/sec CNT100;
   1:  PR[GP1:91,1] = PR[GP1:90,1] + -9.271;
   1:  PR[GP1:91,2] = PR[GP1:90,2] + -24.317;
   1:L PR[91] R[100]mm/sec CNT100;
   1:  PR[GP1:91,1] = PR[GP1:90,1] + -6.905;
   1:  PR[GP1:91,2] = PR[GP1:90,2] + -21.548;
   1:L PR[91] R[100]mm/sec CNT100;
   1:  PR[GP1:91,1] = PR[GP1:90,1] + -4.308;
   1:  PR[GP1:91,2] = PR[GP1:90,2] + -17.998;
   1:L PR[91] R[100]mm/sec CNT100;
   1:  PR[GP1:91,1] = PR[GP1:90,1] + -3.516;
   1:  PR[GP1:91,2] = PR[GP1:90,2] + -17.108;
   1:L PR[91] R[100]mm/sec CNT100;
   1:  PR[GP1:91,1] = PR[GP1:90,1] + -0.683;
   1:  PR[GP1:91,2] = PR[GP1:90,2] + -15.451;
   1:L PR[91] R[100]mm/sec CNT100;
   1:  PR[GP1:91,1] = PR[GP1:90,1] + 0.991;
   1:  PR[GP1:91,2] = PR[GP1:90,2] + -15.435;
   1:L PR[91] R[100]mm/sec CNT100;
   1:  PR[GP1:91,1] = PR[GP1:90,1] + 1.816;
   1:  PR[GP1:91,2] = PR[GP1:90,2] + -16.423;
   1:L PR[91] R[100]mm/sec CNT100;
   1:  PR[GP1:91,1] = PR[GP1:90,1] + 2.214;
   1:  PR[GP1:91,2] = PR[GP1:90,2] + -16.674;
   1:L PR[91] R[100]mm/sec CNT100;
   1:  PR[GP1:91,1] = PR[GP1:90,1] + 4.467;
   1:  PR[GP1:91,2] = PR[GP1:90,2] + -17.908;
   1:L PR[91] R[100]mm/sec CNT100;
   1:  PR[GP1:91,1] = PR[GP1:90,1] + 7.128;
   1:  PR[GP1:91,2] = PR[GP1:90,2] + -21.549;
   1:L PR[91] R[100]mm/sec CNT100;
   1:  PR[GP1:91,1] = PR[GP1:90,1] + 9.502;
   1:  PR[GP1:91,2] = PR[GP1:90,2] + -24.331;
   1:L PR[91] R[100]mm/sec CNT100;
   1:  PR[GP1:91,1] = PR[GP1:90,1] + 15.329;
   1:  PR[GP1:91,2] = PR[GP1:90,2] + -28.644;
   1:L PR[91] R[100]mm/sec CNT100;
   1:  PR[GP1:91,1] = PR[GP1:90,1] + 17.200;
   1:  PR[GP1:91,2] = PR[GP1:90,2] + -30.104;
   1:L PR[91] R[100]mm/sec CNT100;
   1:  PR[GP1:91,1] = PR[GP1:90,1] + 18.589;
   1:  PR[GP1:91,2] = PR[GP1:90,2] + -30.859;
   1:L PR[91] R[100]mm/sec CNT100;
   1:  PR[GP1:91,1] = PR[GP1:90,1] + 27.731;
   1:  PR[GP1:91,2] = PR[GP1:90,2] + -34.078;
   1:L PR[91] R[100]mm/sec CNT100;
   1:  PR[GP1:91,1] = PR[GP1:90,1] + 28.316;
   1:  PR[GP1:91,2] = PR[GP1:90,2] + -34.301;
   1:L PR[91] R[100]mm/sec CNT100;
   1:  PR[GP1:91,1] = PR[GP1:90,1] + 28.418;
   1:  PR[GP1:91,2] = PR[GP1:90,2] + -34.316;
   1:L PR[91] R[100]mm/sec CNT100;
   1:  PR[GP1:91,1] = PR[GP1:90,1] + 38.499;
   1:  PR[GP1:91,2] = PR[GP1:90,2] + -35.035;
   1:L PR[91] R[100]mm/sec CNT100;
   1:  PR[GP1:91,1] = PR[GP1:90,1] + 41.398;
   1:  PR[GP1:91,2] = PR[GP1:90,2] + -34.568;
   1:L PR[91] R[100]mm/sec CNT100;
   1:  PR[GP1:91,1] = PR[GP1:90,1] + 48.743;
   1:  PR[GP1:91,2] = PR[GP1:90,2] + -32.920;
   1:L PR[91] R[100]mm/sec CNT100;
   1:  PR[GP1:91,1] = PR[GP1:90,1] + 53.452;
   1:  PR[GP1:91,2] = PR[GP1:90,2] + -30.556;
   1:L PR[91] R[100]mm/sec CNT100;
   1:  PR[GP1:91,1] = PR[GP1:90,1] + 58.129;
   1:  PR[GP1:91,2] = PR[GP1:90,2] + -27.924;
   1:L PR[91] R[100]mm/sec CNT100;
   1:  PR[GP1:91,1] = PR[GP1:90,1] + 63.089;
   1:  PR[GP1:91,2] = PR[GP1:90,2] + -23.052;
   1:L PR[91] R[100]mm/sec CNT100;
   1:  PR[GP1:91,1] = PR[GP1:90,1] + 65.700;
   1:  PR[GP1:91,2] = PR[GP1:90,2] + -20.293;
   1:L PR[91] R[100]mm/sec CNT100;
   1:  PR[GP1:91,1] = PR[GP1:90,1] + 69.375;
   1:  PR[GP1:91,2] = PR[GP1:90,2] + -13.255;
   1:L PR[91] R[100]mm/sec CNT100;
   1:  PR[GP1:91,1] = PR[GP1:90,1] + 70.621;
   1:  PR[GP1:91,2] = PR[GP1:90,2] + -10.745;
   1:L PR[91] R[100]mm/sec CNT100;
   1:  PR[GP1:91,1] = PR[GP1:90,1] + 71.970;
   1:  PR[GP1:91,2] = PR[GP1:90,2] + -2.421;
   1:L PR[91] R[100]mm/sec CNT100;
   1:  PR[GP1:91,1] = PR[GP1:90,1] + 72.130;
   1:  PR[GP1:91,2] = PR[GP1:90,2] + -1.599;
   1:L PR[91] R[100]mm/sec CNT100;
   1:  PR[GP1:91,1] = PR[GP1:90,1] + 72.363;
   1:  PR[GP1:91,2] = PR[GP1:90,2] + -0.076;
   1:L PR[91] R[100]mm/sec CNT100;
   1:  PR[GP1:91,1] = PR[GP1:90,1] + 70.992;
   1:  PR[GP1:91,2] = PR[GP1:90,2] + 8.161;
   1:L PR[91] R[100]mm/sec CNT100;
   1:  PR[GP1:91,1] = PR[GP1:90,1] + 70.620;
   1:  PR[GP1:91,2] = PR[GP1:90,2] + 10.603;
   1:L PR[91] R[100]mm/sec CNT100;
   1:  PR[GP1:91,1] = PR[GP1:90,1] + 69.375;
   1:  PR[GP1:91,2] = PR[GP1:90,2] + 13.111;
   1:L PR[91] R[100]mm/sec CNT100;
   1:  PR[GP1:91,1] = PR[GP1:90,1] + 65.700;
   1:  PR[GP1:91,2] = PR[GP1:90,2] + 20.149;
   1:L PR[91] R[100]mm/sec CNT100;
   1:  PR[GP1:91,1] = PR[GP1:90,1] + 63.089;
   1:  PR[GP1:91,2] = PR[GP1:90,2] + 22.908;
   1:L PR[91] R[100]mm/sec CNT100;
   1:  PR[GP1:91,1] = PR[GP1:90,1] + 58.129;
   1:  PR[GP1:91,2] = PR[GP1:90,2] + 27.780;
   1:L PR[91] R[100]mm/sec CNT100;
   1:  PR[GP1:91,1] = PR[GP1:90,1] + 53.452;
   1:  PR[GP1:91,2] = PR[GP1:90,2] + 30.412;
   1:L PR[91] R[100]mm/sec CNT100;
   1:  PR[GP1:91,1] = PR[GP1:90,1] + 48.743;
   1:  PR[GP1:91,2] = PR[GP1:90,2] + 32.776;
   1:L PR[91] R[100]mm/sec CNT100;
   1:  PR[GP1:91,1] = PR[GP1:90,1] + 41.398;
   1:  PR[GP1:91,2] = PR[GP1:90,2] + 34.424;
   1:L PR[91] R[100]mm/sec CNT100;
   1:  PR[GP1:91,1] = PR[GP1:90,1] + 38.499;
   1:  PR[GP1:91,2] = PR[GP1:90,2] + 34.891;
   1:L PR[91] R[100]mm/sec CNT100;
   1:  PR[GP1:91,1] = PR[GP1:90,1] + 28.418;
   1:  PR[GP1:91,2] = PR[GP1:90,2] + 34.172;
   1:L PR[91] R[100]mm/sec CNT100;
   1:  PR[GP1:91,1] = PR[GP1:90,1] + 28.316;
   1:  PR[GP1:91,2] = PR[GP1:90,2] + 34.157;
   1:L PR[91] R[100]mm/sec CNT100;
   1:  PR[GP1:91,1] = PR[GP1:90,1] + 27.732;
   1:  PR[GP1:91,2] = PR[GP1:90,2] + 33.935;
   1:L PR[91] R[100]mm/sec CNT100;
   1:  PR[GP1:91,1] = PR[GP1:90,1] + 19.647;
   1:  PR[GP1:91,2] = PR[GP1:90,2] + 31.045;
   1:L PR[91] R[100]mm/sec CNT100;
   1:  PR[GP1:91,1] = PR[GP1:90,1] + 18.580;
   1:  PR[GP1:91,2] = PR[GP1:90,2] + 30.710;
   1:L PR[91] R[100]mm/sec CNT100;
   1:  PR[GP1:91,1] = PR[GP1:90,1] + 17.192;
   1:  PR[GP1:91,2] = PR[GP1:90,2] + 29.955;
   1:L PR[91] R[100]mm/sec CNT100;
   1:  PR[GP1:91,1] = PR[GP1:90,1] + 11.560;
   1:  PR[GP1:91,2] = PR[GP1:90,2] + 25.826;
   1:L PR[91] R[100]mm/sec CNT100;
   1:  PR[GP1:91,1] = PR[GP1:90,1] + 9.509;
   1:  PR[GP1:91,2] = PR[GP1:90,2] + 24.195;
   1:L PR[91] R[100]mm/sec CNT100;
   1:  PR[GP1:91,1] = PR[GP1:90,1] + 7.128;
   1:  PR[GP1:91,2] = PR[GP1:90,2] + 21.405;
   1:L PR[91] R[100]mm/sec CNT100;
   1:  PR[GP1:91,1] = PR[GP1:90,1] + 4.527;
   1:  PR[GP1:91,2] = PR[GP1:90,2] + 17.847;
   1:L PR[91] R[100]mm/sec CNT100;
   1:  PR[GP1:91,1] = PR[GP1:90,1] + 3.712;
   1:  PR[GP1:91,2] = PR[GP1:90,2] + 16.949;
   1:L PR[91] R[100]mm/sec CNT100;
   1:  PR[GP1:91,1] = PR[GP1:90,1] + 0.872;
   1:  PR[GP1:91,2] = PR[GP1:90,2] + 15.292;
   1:L PR[91] R[100]mm/sec CNT100;
   1:  PR[GP1:91,1] = PR[GP1:90,1] + -0.683;
   1:  PR[GP1:91,2] = PR[GP1:90,2] + 15.307;
   1:L PR[91] R[100]mm/sec CNT100;
   1:  ! -- Layer/Ebene 57 -- !;
   1:  PR[91] = PR[90];
   1:  PR[GP1:91,1] = PR[GP1:90,1] + -3.633;
   1:  PR[GP1:91,2] = PR[GP1:90,2] + 17.515;
   1:  PR[GP1:91,3] = PR[GP1:90,3] + 35.075;
   1:L PR[91] R[100]mm/sec CNT100;
   1:  PR[GP1:91,1] = PR[GP1:90,1] + -4.377;
   1:  PR[GP1:91,2] = PR[GP1:90,2] + 18.317;
   1:L PR[91] R[100]mm/sec CNT100;
   1:  PR[GP1:91,1] = PR[GP1:90,1] + -4.384;
   1:  PR[GP1:91,2] = PR[GP1:90,2] + 18.383;
   1:L PR[91] R[100]mm/sec CNT100;
   1:  PR[GP1:91,1] = PR[GP1:90,1] + -6.292;
   1:  PR[GP1:91,2] = PR[GP1:90,2] + 20.991;
   1:L PR[91] R[100]mm/sec CNT100;
   1:  PR[GP1:91,1] = PR[GP1:90,1] + -9.069;
   1:  PR[GP1:91,2] = PR[GP1:90,2] + 24.241;
   1:L PR[91] R[100]mm/sec CNT100;
   1:  PR[GP1:91,1] = PR[GP1:90,1] + -13.958;
   1:  PR[GP1:91,2] = PR[GP1:90,2] + 27.858;
   1:L PR[91] R[100]mm/sec CNT100;
   1:  PR[GP1:91,1] = PR[GP1:90,1] + -16.477;
   1:  PR[GP1:91,2] = PR[GP1:90,2] + 29.825;
   1:L PR[91] R[100]mm/sec CNT100;
   1:  PR[GP1:91,1] = PR[GP1:90,1] + -18.362;
   1:  PR[GP1:91,2] = PR[GP1:90,2] + 30.852;
   1:L PR[91] R[100]mm/sec CNT100;
   1:  PR[GP1:91,1] = PR[GP1:90,1] + -27.422;
   1:  PR[GP1:91,2] = PR[GP1:90,2] + 34.047;
   1:L PR[91] R[100]mm/sec CNT100;
   1:  PR[GP1:91,1] = PR[GP1:90,1] + -27.866;
   1:  PR[GP1:91,2] = PR[GP1:90,2] + 34.192;
   1:L PR[91] R[100]mm/sec CNT100;
   1:  PR[GP1:91,1] = PR[GP1:90,1] + -28.133;
   1:  PR[GP1:91,2] = PR[GP1:90,2] + 34.230;
   1:L PR[91] R[100]mm/sec CNT100;
   1:  PR[GP1:91,1] = PR[GP1:90,1] + -30.341;
   1:  PR[GP1:91,2] = PR[GP1:90,2] + 34.342;
   1:L PR[91] R[100]mm/sec CNT100;
   1:  PR[GP1:91,1] = PR[GP1:90,1] + -38.322;
   1:  PR[GP1:91,2] = PR[GP1:90,2] + 34.910;
   1:L PR[91] R[100]mm/sec CNT100;
   1:  PR[GP1:91,1] = PR[GP1:90,1] + -40.419;
   1:  PR[GP1:91,2] = PR[GP1:90,2] + 34.572;
   1:L PR[91] R[100]mm/sec CNT100;
   1:  PR[GP1:91,1] = PR[GP1:90,1] + -48.526;
   1:  PR[GP1:91,2] = PR[GP1:90,2] + 32.756;
   1:L PR[91] R[100]mm/sec CNT100;
   1:  PR[GP1:91,1] = PR[GP1:90,1] + -52.564;
   1:  PR[GP1:91,2] = PR[GP1:90,2] + 30.726;
   1:L PR[91] R[100]mm/sec CNT100;
   1:  PR[GP1:91,1] = PR[GP1:90,1] + -57.869;
   1:  PR[GP1:91,2] = PR[GP1:90,2] + 27.735;
   1:L PR[91] R[100]mm/sec CNT100;
   1:  PR[GP1:91,1] = PR[GP1:90,1] + -62.335;
   1:  PR[GP1:91,2] = PR[GP1:90,2] + 23.354;
   1:L PR[91] R[100]mm/sec CNT100;
   1:  PR[GP1:91,1] = PR[GP1:90,1] + -65.403;
   1:  PR[GP1:91,2] = PR[GP1:90,2] + 20.122;
   1:L PR[91] R[100]mm/sec CNT100;
   1:  PR[GP1:91,1] = PR[GP1:90,1] + -68.782;
   1:  PR[GP1:91,2] = PR[GP1:90,2] + 13.634;
   1:L PR[91] R[100]mm/sec CNT100;
   1:  PR[GP1:91,1] = PR[GP1:90,1] + -70.300;
   1:  PR[GP1:91,2] = PR[GP1:90,2] + 10.560;
   1:L PR[91] R[100]mm/sec CNT100;
   1:  PR[GP1:91,1] = PR[GP1:90,1] + -71.552;
   1:  PR[GP1:91,2] = PR[GP1:90,2] + 2.844;
   1:L PR[91] R[100]mm/sec CNT100;
   1:  PR[GP1:91,1] = PR[GP1:90,1] + -71.701;
   1:  PR[GP1:91,2] = PR[GP1:90,2] + 2.083;
   1:L PR[91] R[100]mm/sec CNT100;
   1:  PR[GP1:91,1] = PR[GP1:90,1] + -72.030;
   1:  PR[GP1:91,2] = PR[GP1:90,2] + -0.068;
   1:L PR[91] R[100]mm/sec CNT100;
   1:  PR[GP1:91,1] = PR[GP1:90,1] + -70.752;
   1:  PR[GP1:91,2] = PR[GP1:90,2] + -7.737;
   1:L PR[91] R[100]mm/sec CNT100;
   1:  PR[GP1:91,1] = PR[GP1:90,1] + -70.299;
   1:  PR[GP1:91,2] = PR[GP1:90,2] + -10.706;
   1:L PR[91] R[100]mm/sec CNT100;
   1:  PR[GP1:91,1] = PR[GP1:90,1] + -68.782;
   1:  PR[GP1:91,2] = PR[GP1:90,2] + -13.778;
   1:L PR[91] R[100]mm/sec CNT100;
   1:  PR[GP1:91,1] = PR[GP1:90,1] + -65.403;
   1:  PR[GP1:91,2] = PR[GP1:90,2] + -20.266;
   1:L PR[91] R[100]mm/sec CNT100;
   1:  PR[GP1:91,1] = PR[GP1:90,1] + -62.335;
   1:  PR[GP1:91,2] = PR[GP1:90,2] + -23.498;
   1:L PR[91] R[100]mm/sec CNT100;
   1:  PR[GP1:91,1] = PR[GP1:90,1] + -57.869;
   1:  PR[GP1:91,2] = PR[GP1:90,2] + -27.879;
   1:L PR[91] R[100]mm/sec CNT100;
   1:  PR[GP1:91,1] = PR[GP1:90,1] + -52.564;
   1:  PR[GP1:91,2] = PR[GP1:90,2] + -30.870;
   1:L PR[91] R[100]mm/sec CNT100;
   1:  PR[GP1:91,1] = PR[GP1:90,1] + -48.526;
   1:  PR[GP1:91,2] = PR[GP1:90,2] + -32.900;
   1:L PR[91] R[100]mm/sec CNT100;
   1:  PR[GP1:91,1] = PR[GP1:90,1] + -40.419;
   1:  PR[GP1:91,2] = PR[GP1:90,2] + -34.716;
   1:L PR[91] R[100]mm/sec CNT100;
   1:  PR[GP1:91,1] = PR[GP1:90,1] + -38.322;
   1:  PR[GP1:91,2] = PR[GP1:90,2] + -35.054;
   1:L PR[91] R[100]mm/sec CNT100;
   1:  PR[GP1:91,1] = PR[GP1:90,1] + -30.341;
   1:  PR[GP1:91,2] = PR[GP1:90,2] + -34.486;
   1:L PR[91] R[100]mm/sec CNT100;
   1:  PR[GP1:91,1] = PR[GP1:90,1] + -28.133;
   1:  PR[GP1:91,2] = PR[GP1:90,2] + -34.374;
   1:L PR[91] R[100]mm/sec CNT100;
   1:  PR[GP1:91,1] = PR[GP1:90,1] + -27.875;
   1:  PR[GP1:91,2] = PR[GP1:90,2] + -34.337;
   1:L PR[91] R[100]mm/sec CNT100;
   1:  PR[GP1:91,1] = PR[GP1:90,1] + -19.782;
   1:  PR[GP1:91,2] = PR[GP1:90,2] + -31.440;
   1:L PR[91] R[100]mm/sec CNT100;
   1:  PR[GP1:91,1] = PR[GP1:90,1] + -18.353;
   1:  PR[GP1:91,2] = PR[GP1:90,2] + -30.991;
   1:L PR[91] R[100]mm/sec CNT100;
   1:  PR[GP1:91,1] = PR[GP1:90,1] + -16.469;
   1:  PR[GP1:91,2] = PR[GP1:90,2] + -29.964;
   1:L PR[91] R[100]mm/sec CNT100;
   1:  PR[GP1:91,1] = PR[GP1:90,1] + -11.512;
   1:  PR[GP1:91,2] = PR[GP1:90,2] + -26.333;
   1:L PR[91] R[100]mm/sec CNT100;
   1:  PR[GP1:91,1] = PR[GP1:90,1] + -9.076;
   1:  PR[GP1:91,2] = PR[GP1:90,2] + -24.393;
   1:L PR[91] R[100]mm/sec CNT100;
   1:  PR[GP1:91,1] = PR[GP1:90,1] + -6.292;
   1:  PR[GP1:91,2] = PR[GP1:90,2] + -21.135;
   1:L PR[91] R[100]mm/sec CNT100;
   1:  PR[GP1:91,1] = PR[GP1:90,1] + -4.273;
   1:  PR[GP1:91,2] = PR[GP1:90,2] + -18.374;
   1:L PR[91] R[100]mm/sec CNT100;
   1:  PR[GP1:91,1] = PR[GP1:90,1] + -3.639;
   1:  PR[GP1:91,2] = PR[GP1:90,2] + -17.662;
   1:L PR[91] R[100]mm/sec CNT100;
   1:  PR[GP1:91,1] = PR[GP1:90,1] + -0.580;
   1:  PR[GP1:91,2] = PR[GP1:90,2] + -15.873;
   1:L PR[91] R[100]mm/sec CNT100;
   1:  PR[GP1:91,1] = PR[GP1:90,1] + 0.893;
   1:  PR[GP1:91,2] = PR[GP1:90,2] + -15.859;
   1:L PR[91] R[100]mm/sec CNT100;
   1:  PR[GP1:91,1] = PR[GP1:90,1] + 1.602;
   1:  PR[GP1:91,2] = PR[GP1:90,2] + -16.709;
   1:L PR[91] R[100]mm/sec CNT100;
   1:  PR[GP1:91,1] = PR[GP1:90,1] + 1.919;
   1:  PR[GP1:91,2] = PR[GP1:90,2] + -16.908;
   1:L PR[91] R[100]mm/sec CNT100;
   1:  PR[GP1:91,1] = PR[GP1:90,1] + 4.433;
   1:  PR[GP1:91,2] = PR[GP1:90,2] + -18.285;
   1:L PR[91] R[100]mm/sec CNT100;
   1:  PR[GP1:91,1] = PR[GP1:90,1] + 6.517;
   1:  PR[GP1:91,2] = PR[GP1:90,2] + -21.136;
   1:L PR[91] R[100]mm/sec CNT100;
   1:  PR[GP1:91,1] = PR[GP1:90,1] + 9.312;
   1:  PR[GP1:91,2] = PR[GP1:90,2] + -24.411;
   1:L PR[91] R[100]mm/sec CNT100;
   1:  PR[GP1:91,1] = PR[GP1:90,1] + 14.202;
   1:  PR[GP1:91,2] = PR[GP1:90,2] + -28.031;
   1:L PR[91] R[100]mm/sec CNT100;
   1:  PR[GP1:91,1] = PR[GP1:90,1] + 16.698;
   1:  PR[GP1:91,2] = PR[GP1:90,2] + -29.979;
   1:L PR[91] R[100]mm/sec CNT100;
   1:  PR[GP1:91,1] = PR[GP1:90,1] + 18.571;
   1:  PR[GP1:91,2] = PR[GP1:90,2] + -30.997;
   1:L PR[91] R[100]mm/sec CNT100;
   1:  PR[GP1:91,1] = PR[GP1:90,1] + 27.634;
   1:  PR[GP1:91,2] = PR[GP1:90,2] + -34.189;
   1:L PR[91] R[100]mm/sec CNT100;
   1:  PR[GP1:91,1] = PR[GP1:90,1] + 28.080;
   1:  PR[GP1:91,2] = PR[GP1:90,2] + -34.334;
   1:L PR[91] R[100]mm/sec CNT100;
   1:  PR[GP1:91,1] = PR[GP1:90,1] + 28.346;
   1:  PR[GP1:91,2] = PR[GP1:90,2] + -34.373;
   1:L PR[91] R[100]mm/sec CNT100;
   1:  PR[GP1:91,1] = PR[GP1:90,1] + 30.554;
   1:  PR[GP1:91,2] = PR[GP1:90,2] + -34.485;
   1:L PR[91] R[100]mm/sec CNT100;
   1:  PR[GP1:91,1] = PR[GP1:90,1] + 38.534;
   1:  PR[GP1:91,2] = PR[GP1:90,2] + -35.054;
   1:L PR[91] R[100]mm/sec CNT100;
   1:  PR[GP1:91,1] = PR[GP1:90,1] + 40.631;
   1:  PR[GP1:91,2] = PR[GP1:90,2] + -34.717;
   1:L PR[91] R[100]mm/sec CNT100;
   1:  PR[GP1:91,1] = PR[GP1:90,1] + 48.736;
   1:  PR[GP1:91,2] = PR[GP1:90,2] + -32.899;
   1:L PR[91] R[100]mm/sec CNT100;
   1:  PR[GP1:91,1] = PR[GP1:90,1] + 52.775;
   1:  PR[GP1:91,2] = PR[GP1:90,2] + -30.871;
   1:L PR[91] R[100]mm/sec CNT100;
   1:  PR[GP1:91,1] = PR[GP1:90,1] + 58.079;
   1:  PR[GP1:91,2] = PR[GP1:90,2] + -27.886;
   1:L PR[91] R[100]mm/sec CNT100;
   1:  PR[GP1:91,1] = PR[GP1:90,1] + 62.546;
   1:  PR[GP1:91,2] = PR[GP1:90,2] + -23.498;
   1:L PR[91] R[100]mm/sec CNT100;
   1:  PR[GP1:91,1] = PR[GP1:90,1] + 65.615;
   1:  PR[GP1:91,2] = PR[GP1:90,2] + -20.256;
   1:L PR[91] R[100]mm/sec CNT100;
   1:  PR[GP1:91,1] = PR[GP1:90,1] + 68.995;
   1:  PR[GP1:91,2] = PR[GP1:90,2] + -13.783;
   1:L PR[91] R[100]mm/sec CNT100;
   1:  PR[GP1:91,1] = PR[GP1:90,1] + 70.513;
   1:  PR[GP1:91,2] = PR[GP1:90,2] + -10.724;
   1:L PR[91] R[100]mm/sec CNT100;
   1:  PR[GP1:91,1] = PR[GP1:90,1] + 71.765;
   1:  PR[GP1:91,2] = PR[GP1:90,2] + -2.997;
   1:L PR[91] R[100]mm/sec CNT100;
   1:  PR[GP1:91,1] = PR[GP1:90,1] + 71.914;
   1:  PR[GP1:91,2] = PR[GP1:90,2] + -2.234;
   1:L PR[91] R[100]mm/sec CNT100;
   1:  PR[GP1:91,1] = PR[GP1:90,1] + 72.244;
   1:  PR[GP1:91,2] = PR[GP1:90,2] + -0.076;
   1:L PR[91] R[100]mm/sec CNT100;
   1:  PR[GP1:91,1] = PR[GP1:90,1] + 70.965;
   1:  PR[GP1:91,2] = PR[GP1:90,2] + 7.606;
   1:L PR[91] R[100]mm/sec CNT100;
   1:  PR[GP1:91,1] = PR[GP1:90,1] + 70.512;
   1:  PR[GP1:91,2] = PR[GP1:90,2] + 10.583;
   1:L PR[91] R[100]mm/sec CNT100;
   1:  PR[GP1:91,1] = PR[GP1:90,1] + 68.995;
   1:  PR[GP1:91,2] = PR[GP1:90,2] + 13.639;
   1:L PR[91] R[100]mm/sec CNT100;
   1:  PR[GP1:91,1] = PR[GP1:90,1] + 65.615;
   1:  PR[GP1:91,2] = PR[GP1:90,2] + 20.112;
   1:L PR[91] R[100]mm/sec CNT100;
   1:  PR[GP1:91,1] = PR[GP1:90,1] + 62.545;
   1:  PR[GP1:91,2] = PR[GP1:90,2] + 23.354;
   1:L PR[91] R[100]mm/sec CNT100;
   1:  PR[GP1:91,1] = PR[GP1:90,1] + 58.079;
   1:  PR[GP1:91,2] = PR[GP1:90,2] + 27.742;
   1:L PR[91] R[100]mm/sec CNT100;
   1:  PR[GP1:91,1] = PR[GP1:90,1] + 52.775;
   1:  PR[GP1:91,2] = PR[GP1:90,2] + 30.727;
   1:L PR[91] R[100]mm/sec CNT100;
   1:  PR[GP1:91,1] = PR[GP1:90,1] + 48.736;
   1:  PR[GP1:91,2] = PR[GP1:90,2] + 32.755;
   1:L PR[91] R[100]mm/sec CNT100;
   1:  PR[GP1:91,1] = PR[GP1:90,1] + 40.631;
   1:  PR[GP1:91,2] = PR[GP1:90,2] + 34.573;
   1:L PR[91] R[100]mm/sec CNT100;
   1:  PR[GP1:91,1] = PR[GP1:90,1] + 38.534;
   1:  PR[GP1:91,2] = PR[GP1:90,2] + 34.910;
   1:L PR[91] R[100]mm/sec CNT100;
   1:  PR[GP1:91,1] = PR[GP1:90,1] + 30.554;
   1:  PR[GP1:91,2] = PR[GP1:90,2] + 34.341;
   1:L PR[91] R[100]mm/sec CNT100;
   1:  PR[GP1:91,1] = PR[GP1:90,1] + 28.346;
   1:  PR[GP1:91,2] = PR[GP1:90,2] + 34.229;
   1:L PR[91] R[100]mm/sec CNT100;
   1:  PR[GP1:91,1] = PR[GP1:90,1] + 28.089;
   1:  PR[GP1:91,2] = PR[GP1:90,2] + 34.191;
   1:L PR[91] R[100]mm/sec CNT100;
   1:  PR[GP1:91,1] = PR[GP1:90,1] + 19.994;
   1:  PR[GP1:91,2] = PR[GP1:90,2] + 31.298;
   1:L PR[91] R[100]mm/sec CNT100;
   1:  PR[GP1:91,1] = PR[GP1:90,1] + 18.562;
   1:  PR[GP1:91,2] = PR[GP1:90,2] + 30.848;
   1:L PR[91] R[100]mm/sec CNT100;
   1:  PR[GP1:91,1] = PR[GP1:90,1] + 16.691;
   1:  PR[GP1:91,2] = PR[GP1:90,2] + 29.830;
   1:L PR[91] R[100]mm/sec CNT100;
   1:  PR[GP1:91,1] = PR[GP1:90,1] + 11.734;
   1:  PR[GP1:91,2] = PR[GP1:90,2] + 26.196;
   1:L PR[91] R[100]mm/sec CNT100;
   1:  PR[GP1:91,1] = PR[GP1:90,1] + 9.319;
   1:  PR[GP1:91,2] = PR[GP1:90,2] + 24.275;
   1:L PR[91] R[100]mm/sec CNT100;
   1:  PR[GP1:91,1] = PR[GP1:90,1] + 6.517;
   1:  PR[GP1:91,2] = PR[GP1:90,2] + 20.992;
   1:L PR[91] R[100]mm/sec CNT100;
   1:  PR[GP1:91,1] = PR[GP1:90,1] + 4.493;
   1:  PR[GP1:91,2] = PR[GP1:90,2] + 18.224;
   1:L PR[91] R[100]mm/sec CNT100;
   1:  PR[GP1:91,1] = PR[GP1:90,1] + 3.841;
   1:  PR[GP1:91,2] = PR[GP1:90,2] + 17.506;
   1:L PR[91] R[100]mm/sec CNT100;
   1:  PR[GP1:91,1] = PR[GP1:90,1] + 0.774;
   1:  PR[GP1:91,2] = PR[GP1:90,2] + 15.716;
   1:L PR[91] R[100]mm/sec CNT100;
   1:  PR[GP1:91,1] = PR[GP1:90,1] + -0.579;
   1:  PR[GP1:91,2] = PR[GP1:90,2] + 15.729;
   1:L PR[91] R[100]mm/sec CNT100;
   1:  ! -- Layer/Ebene 58 -- !;
   1:  PR[91] = PR[90];
   1:  PR[GP1:91,1] = PR[GP1:90,1] + -3.756;
   1:  PR[GP1:91,2] = PR[GP1:90,2] + 18.070;
   1:  PR[GP1:91,3] = PR[GP1:90,3] + 35.685;
   1:L PR[91] R[100]mm/sec CNT100;
   1:  PR[GP1:91,1] = PR[GP1:90,1] + -4.232;
   1:  PR[GP1:91,2] = PR[GP1:90,2] + 18.584;
   1:L PR[91] R[100]mm/sec CNT100;
   1:  PR[GP1:91,1] = PR[GP1:90,1] + -5.680;
   1:  PR[GP1:91,2] = PR[GP1:90,2] + 20.579;
   1:L PR[91] R[100]mm/sec CNT100;
   1:  PR[GP1:91,1] = PR[GP1:90,1] + -8.874;
   1:  PR[GP1:91,2] = PR[GP1:90,2] + 24.317;
   1:L PR[91] R[100]mm/sec CNT100;
   1:  PR[GP1:91,1] = PR[GP1:90,1] + -12.824;
   1:  PR[GP1:91,2] = PR[GP1:90,2] + 27.239;
   1:L PR[91] R[100]mm/sec CNT100;
   1:  PR[GP1:91,1] = PR[GP1:90,1] + -15.973;
   1:  PR[GP1:91,2] = PR[GP1:90,2] + 29.698;
   1:L PR[91] R[100]mm/sec CNT100;
   1:  PR[GP1:91,1] = PR[GP1:90,1] + -18.345;
   1:  PR[GP1:91,2] = PR[GP1:90,2] + 30.991;
   1:L PR[91] R[100]mm/sec CNT100;
   1:  PR[GP1:91,1] = PR[GP1:90,1] + -26.482;
   1:  PR[GP1:91,2] = PR[GP1:90,2] + 33.860;
   1:L PR[91] R[100]mm/sec CNT100;
   1:  PR[GP1:91,1] = PR[GP1:90,1] + -27.565;
   1:  PR[GP1:91,2] = PR[GP1:90,2] + 34.213;
   1:L PR[91] R[100]mm/sec CNT100;
   1:  PR[GP1:91,1] = PR[GP1:90,1] + -28.273;
   1:  PR[GP1:91,2] = PR[GP1:90,2] + 34.316;
   1:L PR[91] R[100]mm/sec CNT100;
   1:  PR[GP1:91,1] = PR[GP1:90,1] + -33.333;
   1:  PR[GP1:91,2] = PR[GP1:90,2] + 34.572;
   1:L PR[91] R[100]mm/sec CNT100;
   1:  PR[GP1:91,1] = PR[GP1:90,1] + -38.357;
   1:  PR[GP1:91,2] = PR[GP1:90,2] + 34.929;
   1:L PR[91] R[100]mm/sec CNT100;
   1:  PR[GP1:91,1] = PR[GP1:90,1] + -39.650;
   1:  PR[GP1:91,2] = PR[GP1:90,2] + 34.721;
   1:L PR[91] R[100]mm/sec CNT100;
   1:  PR[GP1:91,1] = PR[GP1:90,1] + -48.518;
   1:  PR[GP1:91,2] = PR[GP1:90,2] + 32.735;
   1:L PR[91] R[100]mm/sec CNT100;
   1:  PR[GP1:91,1] = PR[GP1:90,1] + -51.886;
   1:  PR[GP1:91,2] = PR[GP1:90,2] + 31.041;
   1:L PR[91] R[100]mm/sec CNT100;
   1:  PR[GP1:91,1] = PR[GP1:90,1] + -57.819;
   1:  PR[GP1:91,2] = PR[GP1:90,2] + 27.697;
   1:L PR[91] R[100]mm/sec CNT100;
   1:  PR[GP1:91,1] = PR[GP1:90,1] + -61.792;
   1:  PR[GP1:91,2] = PR[GP1:90,2] + 23.799;
   1:L PR[91] R[100]mm/sec CNT100;
   1:  PR[GP1:91,1] = PR[GP1:90,1] + -65.318;
   1:  PR[GP1:91,2] = PR[GP1:90,2] + 20.085;
   1:L PR[91] R[100]mm/sec CNT100;
   1:  PR[GP1:91,1] = PR[GP1:90,1] + -68.401;
   1:  PR[GP1:91,2] = PR[GP1:90,2] + 14.164;
   1:L PR[91] R[100]mm/sec CNT100;
   1:  PR[GP1:91,1] = PR[GP1:90,1] + -70.192;
   1:  PR[GP1:91,2] = PR[GP1:90,2] + 10.539;
   1:L PR[91] R[100]mm/sec CNT100;
   1:  PR[GP1:91,1] = PR[GP1:90,1] + -71.347;
   1:  PR[GP1:91,2] = PR[GP1:90,2] + 3.418;
   1:L PR[91] R[100]mm/sec CNT100;
   1:  PR[GP1:91,1] = PR[GP1:90,1] + -71.484;
   1:  PR[GP1:91,2] = PR[GP1:90,2] + 2.716;
   1:L PR[91] R[100]mm/sec CNT100;
   1:  PR[GP1:91,1] = PR[GP1:90,1] + -71.911;
   1:  PR[GP1:91,2] = PR[GP1:90,2] + -0.068;
   1:L PR[91] R[100]mm/sec CNT100;
   1:  PR[GP1:91,1] = PR[GP1:90,1] + -70.726;
   1:  PR[GP1:91,2] = PR[GP1:90,2] + -7.182;
   1:L PR[91] R[100]mm/sec CNT100;
   1:  PR[GP1:91,1] = PR[GP1:90,1] + -70.191;
   1:  PR[GP1:91,2] = PR[GP1:90,2] + -10.685;
   1:L PR[91] R[100]mm/sec CNT100;
   1:  PR[GP1:91,1] = PR[GP1:90,1] + -68.401;
   1:  PR[GP1:91,2] = PR[GP1:90,2] + -14.308;
   1:L PR[91] R[100]mm/sec CNT100;
   1:  PR[GP1:91,1] = PR[GP1:90,1] + -65.318;
   1:  PR[GP1:91,2] = PR[GP1:90,2] + -20.229;
   1:L PR[91] R[100]mm/sec CNT100;
   1:  PR[GP1:91,1] = PR[GP1:90,1] + -61.792;
   1:  PR[GP1:91,2] = PR[GP1:90,2] + -23.943;
   1:L PR[91] R[100]mm/sec CNT100;
   1:  PR[GP1:91,1] = PR[GP1:90,1] + -57.819;
   1:  PR[GP1:91,2] = PR[GP1:90,2] + -27.841;
   1:L PR[91] R[100]mm/sec CNT100;
   1:  PR[GP1:91,1] = PR[GP1:90,1] + -51.886;
   1:  PR[GP1:91,2] = PR[GP1:90,2] + -31.185;
   1:L PR[91] R[100]mm/sec CNT100;
   1:  PR[GP1:91,1] = PR[GP1:90,1] + -48.518;
   1:  PR[GP1:91,2] = PR[GP1:90,2] + -32.879;
   1:L PR[91] R[100]mm/sec CNT100;
   1:  PR[GP1:91,1] = PR[GP1:90,1] + -39.650;
   1:  PR[GP1:91,2] = PR[GP1:90,2] + -34.865;
   1:L PR[91] R[100]mm/sec CNT100;
   1:  PR[GP1:91,1] = PR[GP1:90,1] + -38.357;
   1:  PR[GP1:91,2] = PR[GP1:90,2] + -35.073;
   1:L PR[91] R[100]mm/sec CNT100;
   1:  PR[GP1:91,1] = PR[GP1:90,1] + -33.333;
   1:  PR[GP1:91,2] = PR[GP1:90,2] + -34.716;
   1:L PR[91] R[100]mm/sec CNT100;
   1:  PR[GP1:91,1] = PR[GP1:90,1] + -28.273;
   1:  PR[GP1:91,2] = PR[GP1:90,2] + -34.460;
   1:L PR[91] R[100]mm/sec CNT100;
   1:  PR[GP1:91,1] = PR[GP1:90,1] + -27.574;
   1:  PR[GP1:91,2] = PR[GP1:90,2] + -34.358;
   1:L PR[91] R[100]mm/sec CNT100;
   1:  PR[GP1:91,1] = PR[GP1:90,1] + -20.129;
   1:  PR[GP1:91,2] = PR[GP1:90,2] + -31.694;
   1:L PR[91] R[100]mm/sec CNT100;
   1:  PR[GP1:91,1] = PR[GP1:90,1] + -18.336;
   1:  PR[GP1:91,2] = PR[GP1:90,2] + -31.130;
   1:L PR[91] R[100]mm/sec CNT100;
   1:  PR[GP1:91,1] = PR[GP1:90,1] + -15.965;
   1:  PR[GP1:91,2] = PR[GP1:90,2] + -29.837;
   1:L PR[91] R[100]mm/sec CNT100;
   1:  PR[GP1:91,1] = PR[GP1:90,1] + -11.684;
   1:  PR[GP1:91,2] = PR[GP1:90,2] + -26.702;
   1:L PR[91] R[100]mm/sec CNT100;
   1:  PR[GP1:91,1] = PR[GP1:90,1] + -8.882;
   1:  PR[GP1:91,2] = PR[GP1:90,2] + -24.469;
   1:L PR[91] R[100]mm/sec CNT100;
   1:  PR[GP1:91,1] = PR[GP1:90,1] + -5.679;
   1:  PR[GP1:91,2] = PR[GP1:90,2] + -20.722;
   1:L PR[91] R[100]mm/sec CNT100;
   1:  PR[GP1:91,1] = PR[GP1:90,1] + -4.237;
   1:  PR[GP1:91,2] = PR[GP1:90,2] + -18.751;
   1:L PR[91] R[100]mm/sec CNT100;
   1:  PR[GP1:91,1] = PR[GP1:90,1] + -3.761;
   1:  PR[GP1:91,2] = PR[GP1:90,2] + -18.217;
   1:L PR[91] R[100]mm/sec CNT100;
   1:  PR[GP1:91,1] = PR[GP1:90,1] + -0.476;
   1:  PR[GP1:91,2] = PR[GP1:90,2] + -16.295;
   1:L PR[91] R[100]mm/sec CNT100;
   1:  PR[GP1:91,1] = PR[GP1:90,1] + 0.794;
   1:  PR[GP1:91,2] = PR[GP1:90,2] + -16.282;
   1:L PR[91] R[100]mm/sec CNT100;
   1:  PR[GP1:91,1] = PR[GP1:90,1] + 1.388;
   1:  PR[GP1:91,2] = PR[GP1:90,2] + -16.994;
   1:L PR[91] R[100]mm/sec CNT100;
   1:  PR[GP1:91,1] = PR[GP1:90,1] + 1.624;
   1:  PR[GP1:91,2] = PR[GP1:90,2] + -17.143;
   1:L PR[91] R[100]mm/sec CNT100;
   1:  PR[GP1:91,1] = PR[GP1:90,1] + 4.399;
   1:  PR[GP1:91,2] = PR[GP1:90,2] + -18.663;
   1:L PR[91] R[100]mm/sec CNT100;
   1:  PR[GP1:91,1] = PR[GP1:90,1] + 5.905;
   1:  PR[GP1:91,2] = PR[GP1:90,2] + -20.723;
   1:L PR[91] R[100]mm/sec CNT100;
   1:  PR[GP1:91,1] = PR[GP1:90,1] + 9.121;
   1:  PR[GP1:91,2] = PR[GP1:90,2] + -24.491;
   1:L PR[91] R[100]mm/sec CNT100;
   1:  PR[GP1:91,1] = PR[GP1:90,1] + 13.075;
   1:  PR[GP1:91,2] = PR[GP1:90,2] + -27.418;
   1:L PR[91] R[100]mm/sec CNT100;
   1:  PR[GP1:91,1] = PR[GP1:90,1] + 16.197;
   1:  PR[GP1:91,2] = PR[GP1:90,2] + -29.854;
   1:L PR[91] R[100]mm/sec CNT100;
   1:  PR[GP1:91,1] = PR[GP1:90,1] + 18.553;
   1:  PR[GP1:91,2] = PR[GP1:90,2] + -31.135;
   1:L PR[91] R[100]mm/sec CNT100;
   1:  PR[GP1:91,1] = PR[GP1:90,1] + 26.692;
   1:  PR[GP1:91,2] = PR[GP1:90,2] + -34.001;
   1:L PR[91] R[100]mm/sec CNT100;
   1:  PR[GP1:91,1] = PR[GP1:90,1] + 27.778;
   1:  PR[GP1:91,2] = PR[GP1:90,2] + -34.355;
   1:L PR[91] R[100]mm/sec CNT100;
   1:  PR[GP1:91,1] = PR[GP1:90,1] + 28.485;
   1:  PR[GP1:91,2] = PR[GP1:90,2] + -34.458;
   1:L PR[91] R[100]mm/sec CNT100;
   1:  PR[GP1:91,1] = PR[GP1:90,1] + 33.546;
   1:  PR[GP1:91,2] = PR[GP1:90,2] + -34.716;
   1:L PR[91] R[100]mm/sec CNT100;
   1:  PR[GP1:91,1] = PR[GP1:90,1] + 38.569;
   1:  PR[GP1:91,2] = PR[GP1:90,2] + -35.074;
   1:L PR[91] R[100]mm/sec CNT100;
   1:  PR[GP1:91,1] = PR[GP1:90,1] + 39.863;
   1:  PR[GP1:91,2] = PR[GP1:90,2] + -34.866;
   1:L PR[91] R[100]mm/sec CNT100;
   1:  PR[GP1:91,1] = PR[GP1:90,1] + 48.729;
   1:  PR[GP1:91,2] = PR[GP1:90,2] + -32.877;
   1:L PR[91] R[100]mm/sec CNT100;
   1:  PR[GP1:91,1] = PR[GP1:90,1] + 52.097;
   1:  PR[GP1:91,2] = PR[GP1:90,2] + -31.186;
   1:L PR[91] R[100]mm/sec CNT100;
   1:  PR[GP1:91,1] = PR[GP1:90,1] + 58.030;
   1:  PR[GP1:91,2] = PR[GP1:90,2] + -27.847;
   1:L PR[91] R[100]mm/sec CNT100;
   1:  PR[GP1:91,1] = PR[GP1:90,1] + 62.002;
   1:  PR[GP1:91,2] = PR[GP1:90,2] + -23.944;
   1:L PR[91] R[100]mm/sec CNT100;
   1:  PR[GP1:91,1] = PR[GP1:90,1] + 65.529;
   1:  PR[GP1:91,2] = PR[GP1:90,2] + -20.218;
   1:L PR[91] R[100]mm/sec CNT100;
   1:  PR[GP1:91,1] = PR[GP1:90,1] + 68.614;
   1:  PR[GP1:91,2] = PR[GP1:90,2] + -14.312;
   1:L PR[91] R[100]mm/sec CNT100;
   1:  PR[GP1:91,1] = PR[GP1:90,1] + 70.405;
   1:  PR[GP1:91,2] = PR[GP1:90,2] + -10.704;
   1:L PR[91] R[100]mm/sec CNT100;
   1:  PR[GP1:91,1] = PR[GP1:90,1] + 71.560;
   1:  PR[GP1:91,2] = PR[GP1:90,2] + -3.573;
   1:L PR[91] R[100]mm/sec CNT100;
   1:  PR[GP1:91,1] = PR[GP1:90,1] + 71.698;
   1:  PR[GP1:91,2] = PR[GP1:90,2] + -2.868;
   1:L PR[91] R[100]mm/sec CNT100;
   1:  PR[GP1:91,1] = PR[GP1:90,1] + 72.125;
   1:  PR[GP1:91,2] = PR[GP1:90,2] + -0.076;
   1:L PR[91] R[100]mm/sec CNT100;
   1:  PR[GP1:91,1] = PR[GP1:90,1] + 70.938;
   1:  PR[GP1:91,2] = PR[GP1:90,2] + 7.050;
   1:L PR[91] R[100]mm/sec CNT100;
   1:  PR[GP1:91,1] = PR[GP1:90,1] + 70.404;
   1:  PR[GP1:91,2] = PR[GP1:90,2] + 10.563;
   1:L PR[91] R[100]mm/sec CNT100;
   1:  PR[GP1:91,1] = PR[GP1:90,1] + 68.614;
   1:  PR[GP1:91,2] = PR[GP1:90,2] + 14.168;
   1:L PR[91] R[100]mm/sec CNT100;
   1:  PR[GP1:91,1] = PR[GP1:90,1] + 65.529;
   1:  PR[GP1:91,2] = PR[GP1:90,2] + 20.074;
   1:L PR[91] R[100]mm/sec CNT100;
   1:  PR[GP1:91,1] = PR[GP1:90,1] + 62.003;
   1:  PR[GP1:91,2] = PR[GP1:90,2] + 23.800;
   1:L PR[91] R[100]mm/sec CNT100;
   1:  PR[GP1:91,1] = PR[GP1:90,1] + 58.029;
   1:  PR[GP1:91,2] = PR[GP1:90,2] + 27.703;
   1:L PR[91] R[100]mm/sec CNT100;
   1:  PR[GP1:91,1] = PR[GP1:90,1] + 52.097;
   1:  PR[GP1:91,2] = PR[GP1:90,2] + 31.042;
   1:L PR[91] R[100]mm/sec CNT100;
   1:  PR[GP1:91,1] = PR[GP1:90,1] + 48.729;
   1:  PR[GP1:91,2] = PR[GP1:90,2] + 32.733;
   1:L PR[91] R[100]mm/sec CNT100;
   1:  PR[GP1:91,1] = PR[GP1:90,1] + 39.863;
   1:  PR[GP1:91,2] = PR[GP1:90,2] + 34.722;
   1:L PR[91] R[100]mm/sec CNT100;
   1:  PR[GP1:91,1] = PR[GP1:90,1] + 38.569;
   1:  PR[GP1:91,2] = PR[GP1:90,2] + 34.930;
   1:L PR[91] R[100]mm/sec CNT100;
   1:  PR[GP1:91,1] = PR[GP1:90,1] + 33.546;
   1:  PR[GP1:91,2] = PR[GP1:90,2] + 34.572;
   1:L PR[91] R[100]mm/sec CNT100;
   1:  PR[GP1:91,1] = PR[GP1:90,1] + 28.485;
   1:  PR[GP1:91,2] = PR[GP1:90,2] + 34.314;
   1:L PR[91] R[100]mm/sec CNT100;
   1:  PR[GP1:91,1] = PR[GP1:90,1] + 27.787;
   1:  PR[GP1:91,2] = PR[GP1:90,2] + 34.212;
   1:L PR[91] R[100]mm/sec CNT100;
   1:  PR[GP1:91,1] = PR[GP1:90,1] + 20.341;
   1:  PR[GP1:91,2] = PR[GP1:90,2] + 31.551;
   1:L PR[91] R[100]mm/sec CNT100;
   1:  PR[GP1:91,1] = PR[GP1:90,1] + 18.544;
   1:  PR[GP1:91,2] = PR[GP1:90,2] + 30.986;
   1:L PR[91] R[100]mm/sec CNT100;
   1:  PR[GP1:91,1] = PR[GP1:90,1] + 16.189;
   1:  PR[GP1:91,2] = PR[GP1:90,2] + 29.705;
   1:L PR[91] R[100]mm/sec CNT100;
   1:  PR[GP1:91,1] = PR[GP1:90,1] + 11.907;
   1:  PR[GP1:91,2] = PR[GP1:90,2] + 26.567;
   1:L PR[91] R[100]mm/sec CNT100;
   1:  PR[GP1:91,1] = PR[GP1:90,1] + 9.128;
   1:  PR[GP1:91,2] = PR[GP1:90,2] + 24.355;
   1:L PR[91] R[100]mm/sec CNT100;
   1:  PR[GP1:91,1] = PR[GP1:90,1] + 5.905;
   1:  PR[GP1:91,2] = PR[GP1:90,2] + 20.579;
   1:L PR[91] R[100]mm/sec CNT100;
   1:  PR[GP1:91,1] = PR[GP1:90,1] + 4.459;
   1:  PR[GP1:91,2] = PR[GP1:90,2] + 18.601;
   1:L PR[91] R[100]mm/sec CNT100;
   1:  PR[GP1:91,1] = PR[GP1:90,1] + 3.970;
   1:  PR[GP1:91,2] = PR[GP1:90,2] + 18.062;
   1:L PR[91] R[100]mm/sec CNT100;
   1:  PR[GP1:91,1] = PR[GP1:90,1] + 0.675;
   1:  PR[GP1:91,2] = PR[GP1:90,2] + 16.140;
   1:L PR[91] R[100]mm/sec CNT100;
   1:  PR[GP1:91,1] = PR[GP1:90,1] + -0.476;
   1:  PR[GP1:91,2] = PR[GP1:90,2] + 16.151;
   1:L PR[91] R[100]mm/sec CNT100;
   1:  ! -- Layer/Ebene 59 -- !;
   1:  PR[91] = PR[90];
   1:  PR[GP1:91,1] = PR[GP1:90,1] + -3.879;
   1:  PR[GP1:91,2] = PR[GP1:90,2] + 18.624;
   1:  PR[GP1:91,3] = PR[GP1:90,3] + 36.295;
   1:L PR[91] R[100]mm/sec CNT100;
   1:  PR[GP1:91,1] = PR[GP1:90,1] + -4.198;
   1:  PR[GP1:91,2] = PR[GP1:90,2] + 18.968;
   1:L PR[91] R[100]mm/sec CNT100;
   1:  PR[GP1:91,1] = PR[GP1:90,1] + -5.066;
   1:  PR[GP1:91,2] = PR[GP1:90,2] + 20.166;
   1:L PR[91] R[100]mm/sec CNT100;
   1:  PR[GP1:91,1] = PR[GP1:90,1] + -8.680;
   1:  PR[GP1:91,2] = PR[GP1:90,2] + 24.393;
   1:L PR[91] R[100]mm/sec CNT100;
   1:  PR[GP1:91,1] = PR[GP1:90,1] + -11.689;
   1:  PR[GP1:91,2] = PR[GP1:90,2] + 26.620;
   1:L PR[91] R[100]mm/sec CNT100;
   1:  PR[GP1:91,1] = PR[GP1:90,1] + -15.469;
   1:  PR[GP1:91,2] = PR[GP1:90,2] + 29.571;
   1:L PR[91] R[100]mm/sec CNT100;
   1:  PR[GP1:91,1] = PR[GP1:90,1] + -18.328;
   1:  PR[GP1:91,2] = PR[GP1:90,2] + 31.130;
   1:L PR[91] R[100]mm/sec CNT100;
   1:  PR[GP1:91,1] = PR[GP1:90,1] + -25.541;
   1:  PR[GP1:91,2] = PR[GP1:90,2] + 33.673;
   1:L PR[91] R[100]mm/sec CNT100;
   1:  PR[GP1:91,1] = PR[GP1:90,1] + -27.264;
   1:  PR[GP1:91,2] = PR[GP1:90,2] + 34.234;
   1:L PR[91] R[100]mm/sec CNT100;
   1:  PR[GP1:91,1] = PR[GP1:90,1] + -28.413;
   1:  PR[GP1:91,2] = PR[GP1:90,2] + 34.401;
   1:L PR[91] R[100]mm/sec CNT100;
   1:  PR[GP1:91,1] = PR[GP1:90,1] + -36.325;
   1:  PR[GP1:91,2] = PR[GP1:90,2] + 34.802;
   1:L PR[91] R[100]mm/sec CNT100;
   1:  PR[GP1:91,1] = PR[GP1:90,1] + -38.391;
   1:  PR[GP1:91,2] = PR[GP1:90,2] + 34.949;
   1:L PR[91] R[100]mm/sec CNT100;
   1:  PR[GP1:91,1] = PR[GP1:90,1] + -38.882;
   1:  PR[GP1:91,2] = PR[GP1:90,2] + 34.870;
   1:L PR[91] R[100]mm/sec CNT100;
   1:  PR[GP1:91,1] = PR[GP1:90,1] + -48.510;
   1:  PR[GP1:91,2] = PR[GP1:90,2] + 32.714;
   1:L PR[91] R[100]mm/sec CNT100;
   1:  PR[GP1:91,1] = PR[GP1:90,1] + -51.208;
   1:  PR[GP1:91,2] = PR[GP1:90,2] + 31.357;
   1:L PR[91] R[100]mm/sec CNT100;
   1:  PR[GP1:91,1] = PR[GP1:90,1] + -57.769;
   1:  PR[GP1:91,2] = PR[GP1:90,2] + 27.658;
   1:L PR[91] R[100]mm/sec CNT100;
   1:  PR[GP1:91,1] = PR[GP1:90,1] + -61.248;
   1:  PR[GP1:91,2] = PR[GP1:90,2] + 24.245;
   1:L PR[91] R[100]mm/sec CNT100;
   1:  PR[GP1:91,1] = PR[GP1:90,1] + -65.233;
   1:  PR[GP1:91,2] = PR[GP1:90,2] + 20.048;
   1:L PR[91] R[100]mm/sec CNT100;
   1:  PR[GP1:91,1] = PR[GP1:90,1] + -68.020;
   1:  PR[GP1:91,2] = PR[GP1:90,2] + 14.695;
   1:L PR[91] R[100]mm/sec CNT100;
   1:  PR[GP1:91,1] = PR[GP1:90,1] + -70.084;
   1:  PR[GP1:91,2] = PR[GP1:90,2] + 10.518;
   1:L PR[91] R[100]mm/sec CNT100;
   1:  PR[GP1:91,1] = PR[GP1:90,1] + -71.142;
   1:  PR[GP1:91,2] = PR[GP1:90,2] + 3.993;
   1:L PR[91] R[100]mm/sec CNT100;
   1:  PR[GP1:91,1] = PR[GP1:90,1] + -71.268;
   1:  PR[GP1:91,2] = PR[GP1:90,2] + 3.349;
   1:L PR[91] R[100]mm/sec CNT100;
   1:  PR[GP1:91,1] = PR[GP1:90,1] + -71.792;
   1:  PR[GP1:91,2] = PR[GP1:90,2] + -0.068;
   1:L PR[91] R[100]mm/sec CNT100;
   1:  PR[GP1:91,1] = PR[GP1:90,1] + -70.699;
   1:  PR[GP1:91,2] = PR[GP1:90,2] + -6.627;
   1:L PR[91] R[100]mm/sec CNT100;
   1:  PR[GP1:91,1] = PR[GP1:90,1] + -70.083;
   1:  PR[GP1:91,2] = PR[GP1:90,2] + -10.664;
   1:L PR[91] R[100]mm/sec CNT100;
   1:  PR[GP1:91,1] = PR[GP1:90,1] + -68.020;
   1:  PR[GP1:91,2] = PR[GP1:90,2] + -14.839;
   1:L PR[91] R[100]mm/sec CNT100;
   1:  PR[GP1:91,1] = PR[GP1:90,1] + -65.233;
   1:  PR[GP1:91,2] = PR[GP1:90,2] + -20.192;
   1:L PR[91] R[100]mm/sec CNT100;
   1:  PR[GP1:91,1] = PR[GP1:90,1] + -61.248;
   1:  PR[GP1:91,2] = PR[GP1:90,2] + -24.389;
   1:L PR[91] R[100]mm/sec CNT100;
   1:  PR[GP1:91,1] = PR[GP1:90,1] + -57.769;
   1:  PR[GP1:91,2] = PR[GP1:90,2] + -27.802;
   1:L PR[91] R[100]mm/sec CNT100;
   1:  PR[GP1:91,1] = PR[GP1:90,1] + -51.208;
   1:  PR[GP1:91,2] = PR[GP1:90,2] + -31.501;
   1:L PR[91] R[100]mm/sec CNT100;
   1:  PR[GP1:91,1] = PR[GP1:90,1] + -48.510;
   1:  PR[GP1:91,2] = PR[GP1:90,2] + -32.858;
   1:L PR[91] R[100]mm/sec CNT100;
   1:  PR[GP1:91,1] = PR[GP1:90,1] + -38.882;
   1:  PR[GP1:91,2] = PR[GP1:90,2] + -35.014;
   1:L PR[91] R[100]mm/sec CNT100;
   1:  PR[GP1:91,1] = PR[GP1:90,1] + -38.391;
   1:  PR[GP1:91,2] = PR[GP1:90,2] + -35.093;
   1:L PR[91] R[100]mm/sec CNT100;
   1:  PR[GP1:91,1] = PR[GP1:90,1] + -36.325;
   1:  PR[GP1:91,2] = PR[GP1:90,2] + -34.946;
   1:L PR[91] R[100]mm/sec CNT100;
   1:  PR[GP1:91,1] = PR[GP1:90,1] + -28.413;
   1:  PR[GP1:91,2] = PR[GP1:90,2] + -34.545;
   1:L PR[91] R[100]mm/sec CNT100;
   1:  PR[GP1:91,1] = PR[GP1:90,1] + -27.272;
   1:  PR[GP1:91,2] = PR[GP1:90,2] + -34.379;
   1:L PR[91] R[100]mm/sec CNT100;
   1:  PR[GP1:91,1] = PR[GP1:90,1] + -20.476;
   1:  PR[GP1:91,2] = PR[GP1:90,2] + -31.947;
   1:L PR[91] R[100]mm/sec CNT100;
   1:  PR[GP1:91,1] = PR[GP1:90,1] + -18.319;
   1:  PR[GP1:91,2] = PR[GP1:90,2] + -31.269;
   1:L PR[91] R[100]mm/sec CNT100;
   1:  PR[GP1:91,1] = PR[GP1:90,1] + -15.461;
   1:  PR[GP1:91,2] = PR[GP1:90,2] + -29.711;
   1:L PR[91] R[100]mm/sec CNT100;
   1:  PR[GP1:91,1] = PR[GP1:90,1] + -11.856;
   1:  PR[GP1:91,2] = PR[GP1:90,2] + -27.070;
   1:L PR[91] R[100]mm/sec CNT100;
   1:  PR[GP1:91,1] = PR[GP1:90,1] + -8.687;
   1:  PR[GP1:91,2] = PR[GP1:90,2] + -24.545;
   1:L PR[91] R[100]mm/sec CNT100;
   1:  PR[GP1:91,1] = PR[GP1:90,1] + -5.066;
   1:  PR[GP1:91,2] = PR[GP1:90,2] + -20.308;
   1:L PR[91] R[100]mm/sec CNT100;
   1:  PR[GP1:91,1] = PR[GP1:90,1] + -4.202;
   1:  PR[GP1:91,2] = PR[GP1:90,2] + -19.128;
   1:L PR[91] R[100]mm/sec CNT100;
   1:  PR[GP1:91,1] = PR[GP1:90,1] + -3.884;
   1:  PR[GP1:91,2] = PR[GP1:90,2] + -18.771;
   1:L PR[91] R[100]mm/sec CNT100;
   1:  PR[GP1:91,1] = PR[GP1:90,1] + -0.372;
   1:  PR[GP1:91,2] = PR[GP1:90,2] + -16.717;
   1:L PR[91] R[100]mm/sec CNT100;
   1:  PR[GP1:91,1] = PR[GP1:90,1] + 0.696;
   1:  PR[GP1:91,2] = PR[GP1:90,2] + -16.706;
   1:L PR[91] R[100]mm/sec CNT100;
   1:  PR[GP1:91,1] = PR[GP1:90,1] + 1.174;
   1:  PR[GP1:91,2] = PR[GP1:90,2] + -17.279;
   1:L PR[91] R[100]mm/sec CNT100;
   1:  PR[GP1:91,1] = PR[GP1:90,1] + 1.329;
   1:  PR[GP1:91,2] = PR[GP1:90,2] + -17.377;
   1:L PR[91] R[100]mm/sec CNT100;
   1:  PR[GP1:91,1] = PR[GP1:90,1] + 4.365;
   1:  PR[GP1:91,2] = PR[GP1:90,2] + -19.040;
   1:L PR[91] R[100]mm/sec CNT100;
   1:  PR[GP1:91,1] = PR[GP1:90,1] + 5.294;
   1:  PR[GP1:91,2] = PR[GP1:90,2] + -20.310;
   1:L PR[91] R[100]mm/sec CNT100;
   1:  PR[GP1:91,1] = PR[GP1:90,1] + 8.930;
   1:  PR[GP1:91,2] = PR[GP1:90,2] + -24.572;
   1:L PR[91] R[100]mm/sec CNT100;
   1:  PR[GP1:91,1] = PR[GP1:90,1] + 11.948;
   1:  PR[GP1:91,2] = PR[GP1:90,2] + -26.806;
   1:L PR[91] R[100]mm/sec CNT100;
   1:  PR[GP1:91,1] = PR[GP1:90,1] + 15.695;
   1:  PR[GP1:91,2] = PR[GP1:90,2] + -29.729;
   1:L PR[91] R[100]mm/sec CNT100;
   1:  PR[GP1:91,1] = PR[GP1:90,1] + 18.535;
   1:  PR[GP1:91,2] = PR[GP1:90,2] + -31.273;
   1:L PR[91] R[100]mm/sec CNT100;
   1:  PR[GP1:91,1] = PR[GP1:90,1] + 25.749;
   1:  PR[GP1:91,2] = PR[GP1:90,2] + -33.814;
   1:L PR[91] R[100]mm/sec CNT100;
   1:  PR[GP1:91,1] = PR[GP1:90,1] + 27.476;
   1:  PR[GP1:91,2] = PR[GP1:90,2] + -34.376;
   1:L PR[91] R[100]mm/sec CNT100;
   1:  PR[GP1:91,1] = PR[GP1:90,1] + 28.624;
   1:  PR[GP1:91,2] = PR[GP1:90,2] + -34.544;
   1:L PR[91] R[100]mm/sec CNT100;
   1:  PR[GP1:91,1] = PR[GP1:90,1] + 36.539;
   1:  PR[GP1:91,2] = PR[GP1:90,2] + -34.946;
   1:L PR[91] R[100]mm/sec CNT100;
   1:  PR[GP1:91,1] = PR[GP1:90,1] + 38.604;
   1:  PR[GP1:91,2] = PR[GP1:90,2] + -35.094;
   1:L PR[91] R[100]mm/sec CNT100;
   1:  PR[GP1:91,1] = PR[GP1:90,1] + 39.095;
   1:  PR[GP1:91,2] = PR[GP1:90,2] + -35.015;
   1:L PR[91] R[100]mm/sec CNT100;
   1:  PR[GP1:91,1] = PR[GP1:90,1] + 48.722;
   1:  PR[GP1:91,2] = PR[GP1:90,2] + -32.855;
   1:L PR[91] R[100]mm/sec CNT100;
   1:  PR[GP1:91,1] = PR[GP1:90,1] + 51.420;
   1:  PR[GP1:91,2] = PR[GP1:90,2] + -31.501;
   1:L PR[91] R[100]mm/sec CNT100;
   1:  PR[GP1:91,1] = PR[GP1:90,1] + 57.980;
   1:  PR[GP1:91,2] = PR[GP1:90,2] + -27.809;
   1:L PR[91] R[100]mm/sec CNT100;
   1:  PR[GP1:91,1] = PR[GP1:90,1] + 61.460;
   1:  PR[GP1:91,2] = PR[GP1:90,2] + -24.390;
   1:L PR[91] R[100]mm/sec CNT100;
   1:  PR[GP1:91,1] = PR[GP1:90,1] + 65.444;
   1:  PR[GP1:91,2] = PR[GP1:90,2] + -20.181;
   1:L PR[91] R[100]mm/sec CNT100;
   1:  PR[GP1:91,1] = PR[GP1:90,1] + 68.233;
   1:  PR[GP1:91,2] = PR[GP1:90,2] + -14.841;
   1:L PR[91] R[100]mm/sec CNT100;
   1:  PR[GP1:91,1] = PR[GP1:90,1] + 70.297;
   1:  PR[GP1:91,2] = PR[GP1:90,2] + -10.684;
   1:L PR[91] R[100]mm/sec CNT100;
   1:  PR[GP1:91,1] = PR[GP1:90,1] + 71.355;
   1:  PR[GP1:91,2] = PR[GP1:90,2] + -4.149;
   1:L PR[91] R[100]mm/sec CNT100;
   1:  PR[GP1:91,1] = PR[GP1:90,1] + 71.481;
   1:  PR[GP1:91,2] = PR[GP1:90,2] + -3.503;
   1:L PR[91] R[100]mm/sec CNT100;
   1:  PR[GP1:91,1] = PR[GP1:90,1] + 72.005;
   1:  PR[GP1:91,2] = PR[GP1:90,2] + -0.076;
   1:L PR[91] R[100]mm/sec CNT100;
   1:  PR[GP1:91,1] = PR[GP1:90,1] + 70.912;
   1:  PR[GP1:91,2] = PR[GP1:90,2] + 6.495;
   1:L PR[91] R[100]mm/sec CNT100;
   1:  PR[GP1:91,1] = PR[GP1:90,1] + 70.295;
   1:  PR[GP1:91,2] = PR[GP1:90,2] + 10.542;
   1:L PR[91] R[100]mm/sec CNT100;
   1:  PR[GP1:91,1] = PR[GP1:90,1] + 68.233;
   1:  PR[GP1:91,2] = PR[GP1:90,2] + 14.697;
   1:L PR[91] R[100]mm/sec CNT100;
   1:  PR[GP1:91,1] = PR[GP1:90,1] + 65.444;
   1:  PR[GP1:91,2] = PR[GP1:90,2] + 20.037;
   1:L PR[91] R[100]mm/sec CNT100;
   1:  PR[GP1:91,1] = PR[GP1:90,1] + 61.459;
   1:  PR[GP1:91,2] = PR[GP1:90,2] + 24.246;
   1:L PR[91] R[100]mm/sec CNT100;
   1:  PR[GP1:91,1] = PR[GP1:90,1] + 57.980;
   1:  PR[GP1:91,2] = PR[GP1:90,2] + 27.665;
   1:L PR[91] R[100]mm/sec CNT100;
   1:  PR[GP1:91,1] = PR[GP1:90,1] + 51.420;
   1:  PR[GP1:91,2] = PR[GP1:90,2] + 31.357;
   1:L PR[91] R[100]mm/sec CNT100;
   1:  PR[GP1:91,1] = PR[GP1:90,1] + 48.722;
   1:  PR[GP1:91,2] = PR[GP1:90,2] + 32.711;
   1:L PR[91] R[100]mm/sec CNT100;
   1:  PR[GP1:91,1] = PR[GP1:90,1] + 39.095;
   1:  PR[GP1:91,2] = PR[GP1:90,2] + 34.871;
   1:L PR[91] R[100]mm/sec CNT100;
   1:  PR[GP1:91,1] = PR[GP1:90,1] + 38.604;
   1:  PR[GP1:91,2] = PR[GP1:90,2] + 34.950;
   1:L PR[91] R[100]mm/sec CNT100;
   1:  PR[GP1:91,1] = PR[GP1:90,1] + 36.539;
   1:  PR[GP1:91,2] = PR[GP1:90,2] + 34.802;
   1:L PR[91] R[100]mm/sec CNT100;
   1:  PR[GP1:91,1] = PR[GP1:90,1] + 28.624;
   1:  PR[GP1:91,2] = PR[GP1:90,2] + 34.400;
   1:L PR[91] R[100]mm/sec CNT100;
   1:  PR[GP1:91,1] = PR[GP1:90,1] + 27.485;
   1:  PR[GP1:91,2] = PR[GP1:90,2] + 34.233;
   1:L PR[91] R[100]mm/sec CNT100;
   1:  PR[GP1:91,1] = PR[GP1:90,1] + 20.688;
   1:  PR[GP1:91,2] = PR[GP1:90,2] + 31.804;
   1:L PR[91] R[100]mm/sec CNT100;
   1:  PR[GP1:91,1] = PR[GP1:90,1] + 18.526;
   1:  PR[GP1:91,2] = PR[GP1:90,2] + 31.124;
   1:L PR[91] R[100]mm/sec CNT100;
   1:  PR[GP1:91,1] = PR[GP1:90,1] + 15.687;
   1:  PR[GP1:91,2] = PR[GP1:90,2] + 29.580;
   1:L PR[91] R[100]mm/sec CNT100;
   1:  PR[GP1:91,1] = PR[GP1:90,1] + 12.081;
   1:  PR[GP1:91,2] = PR[GP1:90,2] + 26.937;
   1:L PR[91] R[100]mm/sec CNT100;
   1:  PR[GP1:91,1] = PR[GP1:90,1] + 8.937;
   1:  PR[GP1:91,2] = PR[GP1:90,2] + 24.436;
   1:L PR[91] R[100]mm/sec CNT100;
   1:  PR[GP1:91,1] = PR[GP1:90,1] + 5.294;
   1:  PR[GP1:91,2] = PR[GP1:90,2] + 20.166;
   1:L PR[91] R[100]mm/sec CNT100;
   1:  PR[GP1:91,1] = PR[GP1:90,1] + 4.425;
   1:  PR[GP1:91,2] = PR[GP1:90,2] + 18.978;
   1:L PR[91] R[100]mm/sec CNT100;
   1:  PR[GP1:91,1] = PR[GP1:90,1] + 4.099;
   1:  PR[GP1:91,2] = PR[GP1:90,2] + 18.618;
   1:L PR[91] R[100]mm/sec CNT100;
   1:  PR[GP1:91,1] = PR[GP1:90,1] + 0.577;
   1:  PR[GP1:91,2] = PR[GP1:90,2] + 16.563;
   1:L PR[91] R[100]mm/sec CNT100;
   1:  PR[GP1:91,1] = PR[GP1:90,1] + -0.372;
   1:  PR[GP1:91,2] = PR[GP1:90,2] + 16.573;
   1:L PR[91] R[100]mm/sec CNT100;
   1:  ! -- Layer/Ebene 60 -- !;
   1:  PR[91] = PR[90];
   1:  PR[GP1:91,1] = PR[GP1:90,1] + -4.002;
   1:  PR[GP1:91,2] = PR[GP1:90,2] + 19.178;
   1:  PR[GP1:91,3] = PR[GP1:90,3] + 36.905;
   1:L PR[91] R[100]mm/sec CNT100;
   1:  PR[GP1:91,1] = PR[GP1:90,1] + -4.163;
   1:  PR[GP1:91,2] = PR[GP1:90,2] + 19.353;
   1:L PR[91] R[100]mm/sec CNT100;
   1:  PR[GP1:91,1] = PR[GP1:90,1] + -4.453;
   1:  PR[GP1:91,2] = PR[GP1:90,2] + 19.752;
   1:L PR[91] R[100]mm/sec CNT100;
   1:  PR[GP1:91,1] = PR[GP1:90,1] + -8.485;
   1:  PR[GP1:91,2] = PR[GP1:90,2] + 24.469;
   1:L PR[91] R[100]mm/sec CNT100;
   1:  PR[GP1:91,1] = PR[GP1:90,1] + -10.555;
   1:  PR[GP1:91,2] = PR[GP1:90,2] + 26.001;
   1:L PR[91] R[100]mm/sec CNT100;
   1:  PR[GP1:91,1] = PR[GP1:90,1] + -14.965;
   1:  PR[GP1:91,2] = PR[GP1:90,2] + 29.445;
   1:L PR[91] R[100]mm/sec CNT100;
   1:  PR[GP1:91,1] = PR[GP1:90,1] + -18.311;
   1:  PR[GP1:91,2] = PR[GP1:90,2] + 31.269;
   1:L PR[91] R[100]mm/sec CNT100;
   1:  PR[GP1:91,1] = PR[GP1:90,1] + -24.600;
   1:  PR[GP1:91,2] = PR[GP1:90,2] + 33.486;
   1:L PR[91] R[100]mm/sec CNT100;
   1:  PR[GP1:91,1] = PR[GP1:90,1] + -26.962;
   1:  PR[GP1:91,2] = PR[GP1:90,2] + 34.255;
   1:L PR[91] R[100]mm/sec CNT100;
   1:  PR[GP1:91,1] = PR[GP1:90,1] + -28.553;
   1:  PR[GP1:91,2] = PR[GP1:90,2] + 34.486;
   1:L PR[91] R[100]mm/sec CNT100;
   1:  PR[GP1:91,1] = PR[GP1:90,1] + -38.266;
   1:  PR[GP1:91,2] = PR[GP1:90,2] + 34.979;
   1:L PR[91] R[100]mm/sec CNT100;
   1:  PR[GP1:91,1] = PR[GP1:90,1] + -38.334;
   1:  PR[GP1:91,2] = PR[GP1:90,2] + 34.977;
   1:L PR[91] R[100]mm/sec CNT100;
   1:  PR[GP1:91,1] = PR[GP1:90,1] + -48.503;
   1:  PR[GP1:91,2] = PR[GP1:90,2] + 32.692;
   1:L PR[91] R[100]mm/sec CNT100;
   1:  PR[GP1:91,1] = PR[GP1:90,1] + -50.530;
   1:  PR[GP1:91,2] = PR[GP1:90,2] + 31.672;
   1:L PR[91] R[100]mm/sec CNT100;
   1:  PR[GP1:91,1] = PR[GP1:90,1] + -57.719;
   1:  PR[GP1:91,2] = PR[GP1:90,2] + 27.620;
   1:L PR[91] R[100]mm/sec CNT100;
   1:  PR[GP1:91,1] = PR[GP1:90,1] + -60.705;
   1:  PR[GP1:91,2] = PR[GP1:90,2] + 24.690;
   1:L PR[91] R[100]mm/sec CNT100;
   1:  PR[GP1:91,1] = PR[GP1:90,1] + -65.148;
   1:  PR[GP1:91,2] = PR[GP1:90,2] + 20.011;
   1:L PR[91] R[100]mm/sec CNT100;
   1:  PR[GP1:91,1] = PR[GP1:90,1] + -67.639;
   1:  PR[GP1:91,2] = PR[GP1:90,2] + 15.226;
   1:L PR[91] R[100]mm/sec CNT100;
   1:  PR[GP1:91,1] = PR[GP1:90,1] + -69.976;
   1:  PR[GP1:91,2] = PR[GP1:90,2] + 10.497;
   1:L PR[91] R[100]mm/sec CNT100;
   1:  PR[GP1:91,1] = PR[GP1:90,1] + -70.938;
   1:  PR[GP1:91,2] = PR[GP1:90,2] + 4.567;
   1:L PR[91] R[100]mm/sec CNT100;
   1:  PR[GP1:91,1] = PR[GP1:90,1] + -71.052;
   1:  PR[GP1:91,2] = PR[GP1:90,2] + 3.981;
   1:L PR[91] R[100]mm/sec CNT100;
   1:  PR[GP1:91,1] = PR[GP1:90,1] + -71.673;
   1:  PR[GP1:91,2] = PR[GP1:90,2] + -0.068;
   1:L PR[91] R[100]mm/sec CNT100;
   1:  PR[GP1:91,1] = PR[GP1:90,1] + -70.672;
   1:  PR[GP1:91,2] = PR[GP1:90,2] + -6.073;
   1:L PR[91] R[100]mm/sec CNT100;
   1:  PR[GP1:91,1] = PR[GP1:90,1] + -69.974;
   1:  PR[GP1:91,2] = PR[GP1:90,2] + -10.643;
   1:L PR[91] R[100]mm/sec CNT100;
   1:  PR[GP1:91,1] = PR[GP1:90,1] + -67.639;
   1:  PR[GP1:91,2] = PR[GP1:90,2] + -15.369;
   1:L PR[91] R[100]mm/sec CNT100;
   1:  PR[GP1:91,1] = PR[GP1:90,1] + -65.148;
   1:  PR[GP1:91,2] = PR[GP1:90,2] + -20.155;
   1:L PR[91] R[100]mm/sec CNT100;
   1:  PR[GP1:91,1] = PR[GP1:90,1] + -60.705;
   1:  PR[GP1:91,2] = PR[GP1:90,2] + -24.834;
   1:L PR[91] R[100]mm/sec CNT100;
   1:  PR[GP1:91,1] = PR[GP1:90,1] + -57.719;
   1:  PR[GP1:91,2] = PR[GP1:90,2] + -27.764;
   1:L PR[91] R[100]mm/sec CNT100;
   1:  PR[GP1:91,1] = PR[GP1:90,1] + -50.531;
   1:  PR[GP1:91,2] = PR[GP1:90,2] + -31.816;
   1:L PR[91] R[100]mm/sec CNT100;
   1:  PR[GP1:91,1] = PR[GP1:90,1] + -48.502;
   1:  PR[GP1:91,2] = PR[GP1:90,2] + -32.836;
   1:L PR[91] R[100]mm/sec CNT100;
   1:  PR[GP1:91,1] = PR[GP1:90,1] + -38.333;
   1:  PR[GP1:91,2] = PR[GP1:90,2] + -35.121;
   1:L PR[91] R[100]mm/sec CNT100;
   1:  PR[GP1:91,1] = PR[GP1:90,1] + -38.266;
   1:  PR[GP1:91,2] = PR[GP1:90,2] + -35.123;
   1:L PR[91] R[100]mm/sec CNT100;
   1:  PR[GP1:91,1] = PR[GP1:90,1] + -28.552;
   1:  PR[GP1:91,2] = PR[GP1:90,2] + -34.630;
   1:L PR[91] R[100]mm/sec CNT100;
   1:  PR[GP1:91,1] = PR[GP1:90,1] + -26.971;
   1:  PR[GP1:91,2] = PR[GP1:90,2] + -34.400;
   1:L PR[91] R[100]mm/sec CNT100;
   1:  PR[GP1:91,1] = PR[GP1:90,1] + -20.823;
   1:  PR[GP1:91,2] = PR[GP1:90,2] + -32.200;
   1:L PR[91] R[100]mm/sec CNT100;
   1:  PR[GP1:91,1] = PR[GP1:90,1] + -18.302;
   1:  PR[GP1:91,2] = PR[GP1:90,2] + -31.408;
   1:L PR[91] R[100]mm/sec CNT100;
   1:  PR[GP1:91,1] = PR[GP1:90,1] + -14.957;
   1:  PR[GP1:91,2] = PR[GP1:90,2] + -29.584;
   1:L PR[91] R[100]mm/sec CNT100;
   1:  PR[GP1:91,1] = PR[GP1:90,1] + -12.028;
   1:  PR[GP1:91,2] = PR[GP1:90,2] + -27.439;
   1:L PR[91] R[100]mm/sec CNT100;
   1:  PR[GP1:91,1] = PR[GP1:90,1] + -8.492;
   1:  PR[GP1:91,2] = PR[GP1:90,2] + -24.621;
   1:L PR[91] R[100]mm/sec CNT100;
   1:  PR[GP1:91,1] = PR[GP1:90,1] + -4.449;
   1:  PR[GP1:91,2] = PR[GP1:90,2] + -19.891;
   1:L PR[91] R[100]mm/sec CNT100;
   1:  PR[GP1:91,1] = PR[GP1:90,1] + -4.028;
   1:  PR[GP1:91,2] = PR[GP1:90,2] + -19.337;
   1:L PR[91] R[100]mm/sec CNT100;
   1:  PR[GP1:91,1] = PR[GP1:90,1] + -0.269;
   1:  PR[GP1:91,2] = PR[GP1:90,2] + -17.138;
   1:L PR[91] R[100]mm/sec CNT100;
   1:  PR[GP1:91,1] = PR[GP1:90,1] + 0.597;
   1:  PR[GP1:91,2] = PR[GP1:90,2] + -17.130;
   1:L PR[91] R[100]mm/sec CNT100;
   1:  PR[GP1:91,1] = PR[GP1:90,1] + 0.960;
   1:  PR[GP1:91,2] = PR[GP1:90,2] + -17.565;
   1:L PR[91] R[100]mm/sec CNT100;
   1:  PR[GP1:91,1] = PR[GP1:90,1] + 1.034;
   1:  PR[GP1:91,2] = PR[GP1:90,2] + -17.611;
   1:L PR[91] R[100]mm/sec CNT100;
   1:  PR[GP1:91,1] = PR[GP1:90,1] + 4.331;
   1:  PR[GP1:91,2] = PR[GP1:90,2] + -19.417;
   1:L PR[91] R[100]mm/sec CNT100;
   1:  PR[GP1:91,1] = PR[GP1:90,1] + 4.683;
   1:  PR[GP1:91,2] = PR[GP1:90,2] + -19.898;
   1:L PR[91] R[100]mm/sec CNT100;
   1:  PR[GP1:91,1] = PR[GP1:90,1] + 8.740;
   1:  PR[GP1:91,2] = PR[GP1:90,2] + -24.652;
   1:L PR[91] R[100]mm/sec CNT100;
   1:  PR[GP1:91,1] = PR[GP1:90,1] + 10.822;
   1:  PR[GP1:91,2] = PR[GP1:90,2] + -26.193;
   1:L PR[91] R[100]mm/sec CNT100;
   1:  PR[GP1:91,1] = PR[GP1:90,1] + 15.193;
   1:  PR[GP1:91,2] = PR[GP1:90,2] + -29.604;
   1:L PR[91] R[100]mm/sec CNT100;
   1:  PR[GP1:91,1] = PR[GP1:90,1] + 18.517;
   1:  PR[GP1:91,2] = PR[GP1:90,2] + -31.411;
   1:L PR[91] R[100]mm/sec CNT100;
   1:  PR[GP1:91,1] = PR[GP1:90,1] + 24.807;
   1:  PR[GP1:91,2] = PR[GP1:90,2] + -33.626;
   1:L PR[91] R[100]mm/sec CNT100;
   1:  PR[GP1:91,1] = PR[GP1:90,1] + 27.174;
   1:  PR[GP1:91,2] = PR[GP1:90,2] + -34.397;
   1:L PR[91] R[100]mm/sec CNT100;
   1:  PR[GP1:91,1] = PR[GP1:90,1] + 28.763;
   1:  PR[GP1:91,2] = PR[GP1:90,2] + -34.629;
   1:L PR[91] R[100]mm/sec CNT100;
   1:  PR[GP1:91,1] = PR[GP1:90,1] + 38.480;
   1:  PR[GP1:91,2] = PR[GP1:90,2] + -35.123;
   1:L PR[91] R[100]mm/sec CNT100;
   1:  PR[GP1:91,1] = PR[GP1:90,1] + 38.547;
   1:  PR[GP1:91,2] = PR[GP1:90,2] + -35.122;
   1:L PR[91] R[100]mm/sec CNT100;
   1:  PR[GP1:91,1] = PR[GP1:90,1] + 48.714;
   1:  PR[GP1:91,2] = PR[GP1:90,2] + -32.834;
   1:L PR[91] R[100]mm/sec CNT100;
   1:  PR[GP1:91,1] = PR[GP1:90,1] + 50.742;
   1:  PR[GP1:91,2] = PR[GP1:90,2] + -31.815;
   1:L PR[91] R[100]mm/sec CNT100;
   1:  PR[GP1:91,1] = PR[GP1:90,1] + 57.930;
   1:  PR[GP1:91,2] = PR[GP1:90,2] + -27.771;
   1:L PR[91] R[100]mm/sec CNT100;
   1:  PR[GP1:91,1] = PR[GP1:90,1] + 60.916;
   1:  PR[GP1:91,2] = PR[GP1:90,2] + -24.836;
   1:L PR[91] R[100]mm/sec CNT100;
   1:  PR[GP1:91,1] = PR[GP1:90,1] + 65.359;
   1:  PR[GP1:91,2] = PR[GP1:90,2] + -20.143;
   1:L PR[91] R[100]mm/sec CNT100;
   1:  PR[GP1:91,1] = PR[GP1:90,1] + 67.852;
   1:  PR[GP1:91,2] = PR[GP1:90,2] + -15.369;
   1:L PR[91] R[100]mm/sec CNT100;
   1:  PR[GP1:91,1] = PR[GP1:90,1] + 70.188;
   1:  PR[GP1:91,2] = PR[GP1:90,2] + -10.663;
   1:L PR[91] R[100]mm/sec CNT100;
   1:  PR[GP1:91,1] = PR[GP1:90,1] + 71.151;
   1:  PR[GP1:91,2] = PR[GP1:90,2] + -4.725;
   1:L PR[91] R[100]mm/sec CNT100;
   1:  PR[GP1:91,1] = PR[GP1:90,1] + 71.265;
   1:  PR[GP1:91,2] = PR[GP1:90,2] + -4.137;
   1:L PR[91] R[100]mm/sec CNT100;
   1:  PR[GP1:91,1] = PR[GP1:90,1] + 71.886;
   1:  PR[GP1:91,2] = PR[GP1:90,2] + -0.076;
   1:L PR[91] R[100]mm/sec CNT100;
   1:  PR[GP1:91,1] = PR[GP1:90,1] + 70.885;
   1:  PR[GP1:91,2] = PR[GP1:90,2] + 5.939;
   1:L PR[91] R[100]mm/sec CNT100;
   1:  PR[GP1:91,1] = PR[GP1:90,1] + 70.187;
   1:  PR[GP1:91,2] = PR[GP1:90,2] + 10.522;
   1:L PR[91] R[100]mm/sec CNT100;
   1:  PR[GP1:91,1] = PR[GP1:90,1] + 67.852;
   1:  PR[GP1:91,2] = PR[GP1:90,2] + 15.225;
   1:L PR[91] R[100]mm/sec CNT100;
   1:  PR[GP1:91,1] = PR[GP1:90,1] + 65.359;
   1:  PR[GP1:91,2] = PR[GP1:90,2] + 19.999;
   1:L PR[91] R[100]mm/sec CNT100;
   1:  PR[GP1:91,1] = PR[GP1:90,1] + 60.916;
   1:  PR[GP1:91,2] = PR[GP1:90,2] + 24.693;
   1:L PR[91] R[100]mm/sec CNT100;
   1:  PR[GP1:91,1] = PR[GP1:90,1] + 57.930;
   1:  PR[GP1:91,2] = PR[GP1:90,2] + 27.627;
   1:L PR[91] R[100]mm/sec CNT100;
   1:  PR[GP1:91,1] = PR[GP1:90,1] + 50.743;
   1:  PR[GP1:91,2] = PR[GP1:90,2] + 31.671;
   1:L PR[91] R[100]mm/sec CNT100;
   1:  PR[GP1:91,1] = PR[GP1:90,1] + 48.714;
   1:  PR[GP1:91,2] = PR[GP1:90,2] + 32.690;
   1:L PR[91] R[100]mm/sec CNT100;
   1:  PR[GP1:91,1] = PR[GP1:90,1] + 38.547;
   1:  PR[GP1:91,2] = PR[GP1:90,2] + 34.978;
   1:L PR[91] R[100]mm/sec CNT100;
   1:  PR[GP1:91,1] = PR[GP1:90,1] + 38.480;
   1:  PR[GP1:91,2] = PR[GP1:90,2] + 34.979;
   1:L PR[91] R[100]mm/sec CNT100;
   1:  PR[GP1:91,1] = PR[GP1:90,1] + 28.763;
   1:  PR[GP1:91,2] = PR[GP1:90,2] + 34.485;
   1:L PR[91] R[100]mm/sec CNT100;
   1:  PR[GP1:91,1] = PR[GP1:90,1] + 27.183;
   1:  PR[GP1:91,2] = PR[GP1:90,2] + 34.254;
   1:L PR[91] R[100]mm/sec CNT100;
   1:  PR[GP1:91,1] = PR[GP1:90,1] + 21.035;
   1:  PR[GP1:91,2] = PR[GP1:90,2] + 32.057;
   1:L PR[91] R[100]mm/sec CNT100;
   1:  PR[GP1:91,1] = PR[GP1:90,1] + 18.508;
   1:  PR[GP1:91,2] = PR[GP1:90,2] + 31.262;
   1:L PR[91] R[100]mm/sec CNT100;
   1:  PR[GP1:91,1] = PR[GP1:90,1] + 15.185;
   1:  PR[GP1:91,2] = PR[GP1:90,2] + 29.455;
   1:L PR[91] R[100]mm/sec CNT100;
   1:  PR[GP1:91,1] = PR[GP1:90,1] + 12.254;
   1:  PR[GP1:91,2] = PR[GP1:90,2] + 27.307;
   1:L PR[91] R[100]mm/sec CNT100;
   1:  PR[GP1:91,1] = PR[GP1:90,1] + 8.747;
   1:  PR[GP1:91,2] = PR[GP1:90,2] + 24.516;
   1:L PR[91] R[100]mm/sec CNT100;
   1:  PR[GP1:91,1] = PR[GP1:90,1] + 4.683;
   1:  PR[GP1:91,2] = PR[GP1:90,2] + 19.754;
   1:L PR[91] R[100]mm/sec CNT100;
   1:  PR[GP1:91,1] = PR[GP1:90,1] + 4.391;
   1:  PR[GP1:91,2] = PR[GP1:90,2] + 19.355;
   1:L PR[91] R[100]mm/sec CNT100;
   1:  PR[GP1:91,1] = PR[GP1:90,1] + 4.227;
   1:  PR[GP1:91,2] = PR[GP1:90,2] + 19.175;
   1:L PR[91] R[100]mm/sec CNT100;
   1:  PR[GP1:91,1] = PR[GP1:90,1] + 0.478;
   1:  PR[GP1:91,2] = PR[GP1:90,2] + 16.987;
   1:L PR[91] R[100]mm/sec CNT100;
   1:  PR[GP1:91,1] = PR[GP1:90,1] + -0.269;
   1:  PR[GP1:91,2] = PR[GP1:90,2] + 16.994;
   1:L PR[91] R[100]mm/sec CNT100;
   1:  ! -- Layer/Ebene 61 -- !;
   1:  PR[91] = PR[90];
   1:  PR[GP1:91,1] = PR[GP1:90,1] + -2.757;
   1:  PR[GP1:91,2] = PR[GP1:90,2] + 18.932;
   1:  PR[GP1:91,3] = PR[GP1:90,3] + 37.515;
   1:L PR[91] R[100]mm/sec CNT100;
   1:  PR[GP1:91,1] = PR[GP1:90,1] + -4.045;
   1:  PR[GP1:91,2] = PR[GP1:90,2] + 19.588;
   1:L PR[91] R[100]mm/sec CNT100;
   1:  PR[GP1:91,1] = PR[GP1:90,1] + -8.290;
   1:  PR[GP1:91,2] = PR[GP1:90,2] + 24.545;
   1:L PR[91] R[100]mm/sec CNT100;
   1:  PR[GP1:91,1] = PR[GP1:90,1] + -9.420;
   1:  PR[GP1:91,2] = PR[GP1:90,2] + 25.382;
   1:L PR[91] R[100]mm/sec CNT100;
   1:  PR[GP1:91,1] = PR[GP1:90,1] + -14.461;
   1:  PR[GP1:91,2] = PR[GP1:90,2] + 29.318;
   1:L PR[91] R[100]mm/sec CNT100;
   1:  PR[GP1:91,1] = PR[GP1:90,1] + -18.294;
   1:  PR[GP1:91,2] = PR[GP1:90,2] + 31.408;
   1:L PR[91] R[100]mm/sec CNT100;
   1:  PR[GP1:91,1] = PR[GP1:90,1] + -23.660;
   1:  PR[GP1:91,2] = PR[GP1:90,2] + 33.300;
   1:L PR[91] R[100]mm/sec CNT100;
   1:  PR[GP1:91,1] = PR[GP1:90,1] + -26.661;
   1:  PR[GP1:91,2] = PR[GP1:90,2] + 34.276;
   1:L PR[91] R[100]mm/sec CNT100;
   1:  PR[GP1:91,1] = PR[GP1:90,1] + -28.692;
   1:  PR[GP1:91,2] = PR[GP1:90,2] + 34.572;
   1:L PR[91] R[100]mm/sec CNT100;
   1:  PR[GP1:91,1] = PR[GP1:90,1] + -37.615;
   1:  PR[GP1:91,2] = PR[GP1:90,2] + 35.024;
   1:L PR[91] R[100]mm/sec CNT100;
   1:  PR[GP1:91,1] = PR[GP1:90,1] + -38.212;
   1:  PR[GP1:91,2] = PR[GP1:90,2] + 35.007;
   1:L PR[91] R[100]mm/sec CNT100;
   1:  PR[GP1:91,1] = PR[GP1:90,1] + -42.137;
   1:  PR[GP1:91,2] = PR[GP1:90,2] + 34.095;
   1:L PR[91] R[100]mm/sec CNT100;
   1:  PR[GP1:91,1] = PR[GP1:90,1] + -48.495;
   1:  PR[GP1:91,2] = PR[GP1:90,2] + 32.671;
   1:L PR[91] R[100]mm/sec CNT100;
   1:  PR[GP1:91,1] = PR[GP1:90,1] + -49.853;
   1:  PR[GP1:91,2] = PR[GP1:90,2] + 31.988;
   1:L PR[91] R[100]mm/sec CNT100;
   1:  PR[GP1:91,1] = PR[GP1:90,1] + -57.669;
   1:  PR[GP1:91,2] = PR[GP1:90,2] + 27.582;
   1:L PR[91] R[100]mm/sec CNT100;
   1:  PR[GP1:91,1] = PR[GP1:90,1] + -60.162;
   1:  PR[GP1:91,2] = PR[GP1:90,2] + 25.136;
   1:L PR[91] R[100]mm/sec CNT100;
   1:  PR[GP1:91,1] = PR[GP1:90,1] + -65.062;
   1:  PR[GP1:91,2] = PR[GP1:90,2] + 19.974;
   1:L PR[91] R[100]mm/sec CNT100;
   1:  PR[GP1:91,1] = PR[GP1:90,1] + -67.258;
   1:  PR[GP1:91,2] = PR[GP1:90,2] + 15.756;
   1:L PR[91] R[100]mm/sec CNT100;
   1:  PR[GP1:91,1] = PR[GP1:90,1] + -69.867;
   1:  PR[GP1:91,2] = PR[GP1:90,2] + 10.476;
   1:L PR[91] R[100]mm/sec CNT100;
   1:  PR[GP1:91,1] = PR[GP1:90,1] + -70.733;
   1:  PR[GP1:91,2] = PR[GP1:90,2] + 5.142;
   1:L PR[91] R[100]mm/sec CNT100;
   1:  PR[GP1:91,1] = PR[GP1:90,1] + -70.836;
   1:  PR[GP1:91,2] = PR[GP1:90,2] + 4.614;
   1:L PR[91] R[100]mm/sec CNT100;
   1:  PR[GP1:91,1] = PR[GP1:90,1] + -71.554;
   1:  PR[GP1:91,2] = PR[GP1:90,2] + -0.068;
   1:L PR[91] R[100]mm/sec CNT100;
   1:  PR[GP1:91,1] = PR[GP1:90,1] + -70.645;
   1:  PR[GP1:91,2] = PR[GP1:90,2] + -5.518;
   1:L PR[91] R[100]mm/sec CNT100;
   1:  PR[GP1:91,1] = PR[GP1:90,1] + -69.866;
   1:  PR[GP1:91,2] = PR[GP1:90,2] + -10.622;
   1:L PR[91] R[100]mm/sec CNT100;
   1:  PR[GP1:91,1] = PR[GP1:90,1] + -67.258;
   1:  PR[GP1:91,2] = PR[GP1:90,2] + -15.900;
   1:L PR[91] R[100]mm/sec CNT100;
   1:  PR[GP1:91,1] = PR[GP1:90,1] + -65.062;
   1:  PR[GP1:91,2] = PR[GP1:90,2] + -20.118;
   1:L PR[91] R[100]mm/sec CNT100;
   1:  PR[GP1:91,1] = PR[GP1:90,1] + -60.162;
   1:  PR[GP1:91,2] = PR[GP1:90,2] + -25.280;
   1:L PR[91] R[100]mm/sec CNT100;
   1:  PR[GP1:91,1] = PR[GP1:90,1] + -57.669;
   1:  PR[GP1:91,2] = PR[GP1:90,2] + -27.726;
   1:L PR[91] R[100]mm/sec CNT100;
   1:  PR[GP1:91,1] = PR[GP1:90,1] + -49.853;
   1:  PR[GP1:91,2] = PR[GP1:90,2] + -32.132;
   1:L PR[91] R[100]mm/sec CNT100;
   1:  PR[GP1:91,1] = PR[GP1:90,1] + -48.495;
   1:  PR[GP1:91,2] = PR[GP1:90,2] + -32.815;
   1:L PR[91] R[100]mm/sec CNT100;
   1:  PR[GP1:91,1] = PR[GP1:90,1] + -42.137;
   1:  PR[GP1:91,2] = PR[GP1:90,2] + -34.239;
   1:L PR[91] R[100]mm/sec CNT100;
   1:  PR[GP1:91,1] = PR[GP1:90,1] + -38.212;
   1:  PR[GP1:91,2] = PR[GP1:90,2] + -35.151;
   1:L PR[91] R[100]mm/sec CNT100;
   1:  PR[GP1:91,1] = PR[GP1:90,1] + -37.615;
   1:  PR[GP1:91,2] = PR[GP1:90,2] + -35.168;
   1:L PR[91] R[100]mm/sec CNT100;
   1:  PR[GP1:91,1] = PR[GP1:90,1] + -28.692;
   1:  PR[GP1:91,2] = PR[GP1:90,2] + -34.716;
   1:L PR[91] R[100]mm/sec CNT100;
   1:  PR[GP1:91,1] = PR[GP1:90,1] + -26.669;
   1:  PR[GP1:91,2] = PR[GP1:90,2] + -34.422;
   1:L PR[91] R[100]mm/sec CNT100;
   1:  PR[GP1:91,1] = PR[GP1:90,1] + -21.171;
   1:  PR[GP1:91,2] = PR[GP1:90,2] + -32.454;
   1:L PR[91] R[100]mm/sec CNT100;
   1:  PR[GP1:91,1] = PR[GP1:90,1] + -18.285;
   1:  PR[GP1:91,2] = PR[GP1:90,2] + -31.547;
   1:L PR[91] R[100]mm/sec CNT100;
   1:  PR[GP1:91,1] = PR[GP1:90,1] + -14.453;
   1:  PR[GP1:91,2] = PR[GP1:90,2] + -29.457;
   1:L PR[91] R[100]mm/sec CNT100;
   1:  PR[GP1:91,1] = PR[GP1:90,1] + -12.200;
   1:  PR[GP1:91,2] = PR[GP1:90,2] + -27.807;
   1:L PR[91] R[100]mm/sec CNT100;
   1:  PR[GP1:91,1] = PR[GP1:90,1] + -8.297;
   1:  PR[GP1:91,2] = PR[GP1:90,2] + -24.697;
   1:L PR[91] R[100]mm/sec CNT100;
   1:  PR[GP1:91,1] = PR[GP1:90,1] + -3.991;
   1:  PR[GP1:91,2] = PR[GP1:90,2] + -19.671;
   1:L PR[91] R[100]mm/sec CNT100;
   1:  PR[GP1:91,1] = PR[GP1:90,1] + -3.804;
   1:  PR[GP1:91,2] = PR[GP1:90,2] + -19.631;
   1:L PR[91] R[100]mm/sec CNT100;
   1:  PR[GP1:91,1] = PR[GP1:90,1] + -2.761;
   1:  PR[GP1:91,2] = PR[GP1:90,2] + -19.079;
   1:L PR[91] R[100]mm/sec CNT100;
   1:  PR[GP1:91,1] = PR[GP1:90,1] + -0.165;
   1:  PR[GP1:91,2] = PR[GP1:90,2] + -17.560;
   1:L PR[91] R[100]mm/sec CNT100;
   1:  PR[GP1:91,1] = PR[GP1:90,1] + 0.499;
   1:  PR[GP1:91,2] = PR[GP1:90,2] + -17.554;
   1:L PR[91] R[100]mm/sec CNT100;
   1:  PR[GP1:91,1] = PR[GP1:90,1] + 0.745;
   1:  PR[GP1:91,2] = PR[GP1:90,2] + -17.849;
   1:L PR[91] R[100]mm/sec CNT100;
   1:  PR[GP1:91,1] = PR[GP1:90,1] + 2.986;
   1:  PR[GP1:91,2] = PR[GP1:90,2] + -19.076;
   1:L PR[91] R[100]mm/sec CNT100;
   1:  PR[GP1:91,1] = PR[GP1:90,1] + 4.273;
   1:  PR[GP1:91,2] = PR[GP1:90,2] + -19.734;
   1:L PR[91] R[100]mm/sec CNT100;
   1:  PR[GP1:91,1] = PR[GP1:90,1] + 8.549;
   1:  PR[GP1:91,2] = PR[GP1:90,2] + -24.732;
   1:L PR[91] R[100]mm/sec CNT100;
   1:  PR[GP1:91,1] = PR[GP1:90,1] + 9.695;
   1:  PR[GP1:91,2] = PR[GP1:90,2] + -25.580;
   1:L PR[91] R[100]mm/sec CNT100;
   1:  PR[GP1:91,1] = PR[GP1:90,1] + 14.691;
   1:  PR[GP1:91,2] = PR[GP1:90,2] + -29.479;
   1:L PR[91] R[100]mm/sec CNT100;
   1:  PR[GP1:91,1] = PR[GP1:90,1] + 18.499;
   1:  PR[GP1:91,2] = PR[GP1:90,2] + -31.549;
   1:L PR[91] R[100]mm/sec CNT100;
   1:  PR[GP1:91,1] = PR[GP1:90,1] + 23.864;
   1:  PR[GP1:91,2] = PR[GP1:90,2] + -33.439;
   1:L PR[91] R[100]mm/sec CNT100;
   1:  PR[GP1:91,1] = PR[GP1:90,1] + 26.872;
   1:  PR[GP1:91,2] = PR[GP1:90,2] + -34.418;
   1:L PR[91] R[100]mm/sec CNT100;
   1:  PR[GP1:91,1] = PR[GP1:90,1] + 28.902;
   1:  PR[GP1:91,2] = PR[GP1:90,2] + -34.715;
   1:L PR[91] R[100]mm/sec CNT100;
   1:  PR[GP1:91,1] = PR[GP1:90,1] + 37.828;
   1:  PR[GP1:91,2] = PR[GP1:90,2] + -35.169;
   1:L PR[91] R[100]mm/sec CNT100;
   1:  PR[GP1:91,1] = PR[GP1:90,1] + 38.422;
   1:  PR[GP1:91,2] = PR[GP1:90,2] + -35.152;
   1:L PR[91] R[100]mm/sec CNT100;
   1:  PR[GP1:91,1] = PR[GP1:90,1] + 42.350;
   1:  PR[GP1:91,2] = PR[GP1:90,2] + -34.238;
   1:L PR[91] R[100]mm/sec CNT100;
   1:  PR[GP1:91,1] = PR[GP1:90,1] + 48.707;
   1:  PR[GP1:91,2] = PR[GP1:90,2] + -32.812;
   1:L PR[91] R[100]mm/sec CNT100;
   1:  PR[GP1:91,1] = PR[GP1:90,1] + 50.065;
   1:  PR[GP1:91,2] = PR[GP1:90,2] + -32.130;
   1:L PR[91] R[100]mm/sec CNT100;
   1:  PR[GP1:91,1] = PR[GP1:90,1] + 57.880;
   1:  PR[GP1:91,2] = PR[GP1:90,2] + -27.732;
   1:L PR[91] R[100]mm/sec CNT100;
   1:  PR[GP1:91,1] = PR[GP1:90,1] + 60.373;
   1:  PR[GP1:91,2] = PR[GP1:90,2] + -25.283;
   1:L PR[91] R[100]mm/sec CNT100;
   1:  PR[GP1:91,1] = PR[GP1:90,1] + 65.274;
   1:  PR[GP1:91,2] = PR[GP1:90,2] + -20.106;
   1:L PR[91] R[100]mm/sec CNT100;
   1:  PR[GP1:91,1] = PR[GP1:90,1] + 67.471;
   1:  PR[GP1:91,2] = PR[GP1:90,2] + -15.898;
   1:L PR[91] R[100]mm/sec CNT100;
   1:  PR[GP1:91,1] = PR[GP1:90,1] + 70.080;
   1:  PR[GP1:91,2] = PR[GP1:90,2] + -10.643;
   1:L PR[91] R[100]mm/sec CNT100;
   1:  PR[GP1:91,1] = PR[GP1:90,1] + 70.946;
   1:  PR[GP1:91,2] = PR[GP1:90,2] + -5.301;
   1:L PR[91] R[100]mm/sec CNT100;
   1:  PR[GP1:91,1] = PR[GP1:90,1] + 71.049;
   1:  PR[GP1:91,2] = PR[GP1:90,2] + -4.772;
   1:L PR[91] R[100]mm/sec CNT100;
   1:  PR[GP1:91,1] = PR[GP1:90,1] + 71.767;
   1:  PR[GP1:91,2] = PR[GP1:90,2] + -0.076;
   1:L PR[91] R[100]mm/sec CNT100;
   1:  PR[GP1:91,1] = PR[GP1:90,1] + 70.858;
   1:  PR[GP1:91,2] = PR[GP1:90,2] + 5.384;
   1:L PR[91] R[100]mm/sec CNT100;
   1:  PR[GP1:91,1] = PR[GP1:90,1] + 70.079;
   1:  PR[GP1:91,2] = PR[GP1:90,2] + 10.502;
   1:L PR[91] R[100]mm/sec CNT100;
   1:  PR[GP1:91,1] = PR[GP1:90,1] + 67.471;
   1:  PR[GP1:91,2] = PR[GP1:90,2] + 15.754;
   1:L PR[91] R[100]mm/sec CNT100;
   1:  PR[GP1:91,1] = PR[GP1:90,1] + 65.274;
   1:  PR[GP1:91,2] = PR[GP1:90,2] + 19.962;
   1:L PR[91] R[100]mm/sec CNT100;
   1:  PR[GP1:91,1] = PR[GP1:90,1] + 60.373;
   1:  PR[GP1:91,2] = PR[GP1:90,2] + 25.139;
   1:L PR[91] R[100]mm/sec CNT100;
   1:  PR[GP1:91,1] = PR[GP1:90,1] + 57.880;
   1:  PR[GP1:91,2] = PR[GP1:90,2] + 27.588;
   1:L PR[91] R[100]mm/sec CNT100;
   1:  PR[GP1:91,1] = PR[GP1:90,1] + 50.065;
   1:  PR[GP1:91,2] = PR[GP1:90,2] + 31.986;
   1:L PR[91] R[100]mm/sec CNT100;
   1:  PR[GP1:91,1] = PR[GP1:90,1] + 48.707;
   1:  PR[GP1:91,2] = PR[GP1:90,2] + 32.668;
   1:L PR[91] R[100]mm/sec CNT100;
   1:  PR[GP1:91,1] = PR[GP1:90,1] + 42.349;
   1:  PR[GP1:91,2] = PR[GP1:90,2] + 34.094;
   1:L PR[91] R[100]mm/sec CNT100;
   1:  PR[GP1:91,1] = PR[GP1:90,1] + 38.830;
   1:  PR[GP1:91,2] = PR[GP1:90,2] + 34.924;
   1:L PR[91] R[100]mm/sec CNT100;
   1:  PR[GP1:91,1] = PR[GP1:90,1] + 38.428;
   1:  PR[GP1:91,2] = PR[GP1:90,2] + 35.008;
   1:L PR[91] R[100]mm/sec CNT100;
   1:  PR[GP1:91,1] = PR[GP1:90,1] + 37.828;
   1:  PR[GP1:91,2] = PR[GP1:90,2] + 35.025;
   1:L PR[91] R[100]mm/sec CNT100;
   1:  PR[GP1:91,1] = PR[GP1:90,1] + 28.902;
   1:  PR[GP1:91,2] = PR[GP1:90,2] + 34.571;
   1:L PR[91] R[100]mm/sec CNT100;
   1:  PR[GP1:91,1] = PR[GP1:90,1] + 26.881;
   1:  PR[GP1:91,2] = PR[GP1:90,2] + 34.275;
   1:L PR[91] R[100]mm/sec CNT100;
   1:  PR[GP1:91,1] = PR[GP1:90,1] + 21.382;
   1:  PR[GP1:91,2] = PR[GP1:90,2] + 32.310;
   1:L PR[91] R[100]mm/sec CNT100;
   1:  PR[GP1:91,1] = PR[GP1:90,1] + 18.490;
   1:  PR[GP1:91,2] = PR[GP1:90,2] + 31.400;
   1:L PR[91] R[100]mm/sec CNT100;
   1:  PR[GP1:91,1] = PR[GP1:90,1] + 14.684;
   1:  PR[GP1:91,2] = PR[GP1:90,2] + 29.330;
   1:L PR[91] R[100]mm/sec CNT100;
   1:  PR[GP1:91,1] = PR[GP1:90,1] + 12.428;
   1:  PR[GP1:91,2] = PR[GP1:90,2] + 27.677;
   1:L PR[91] R[100]mm/sec CNT100;
   1:  PR[GP1:91,1] = PR[GP1:90,1] + 8.556;
   1:  PR[GP1:91,2] = PR[GP1:90,2] + 24.596;
   1:L PR[91] R[100]mm/sec CNT100;
   1:  PR[GP1:91,1] = PR[GP1:90,1] + 4.272;
   1:  PR[GP1:91,2] = PR[GP1:90,2] + 19.586;
   1:L PR[91] R[100]mm/sec CNT100;
   1:  PR[GP1:91,1] = PR[GP1:90,1] + 2.993;
   1:  PR[GP1:91,2] = PR[GP1:90,2] + 18.936;
   1:L PR[91] R[100]mm/sec CNT100;
   1:  PR[GP1:91,1] = PR[GP1:90,1] + 0.380;
   1:  PR[GP1:91,2] = PR[GP1:90,2] + 17.411;
   1:L PR[91] R[100]mm/sec CNT100;
   1:  PR[GP1:91,1] = PR[GP1:90,1] + -0.165;
   1:  PR[GP1:91,2] = PR[GP1:90,2] + 17.416;
   1:L PR[91] R[100]mm/sec CNT100 TB   .50sec,CALL END_PUD;
   1:  DO[117:Laser Start]=OFF;
   1:  !Sicherheitspunkt!;
   1:  PR[92] = PR[91];
   1:  PR[92] = PR[GP1:92,3] + 50;
   1:J PR[92];
   1:  WAIT   5.00(sec);
   1:  DO[119:Gas]=OFF;
   1:  CALL HOME_ALL;
/POS
/END
